# B&R Automation Studio project TD52 (part 100)

#### gwt.var - Local variables
```iecst
VAR
	xGR_MAXR_FA_AN_LAGA1 : GR_MAXR;
	xGR_MAXR_FA_GWW1 : GR_MAXR;
	xGR_MAXR_FA_AN_LAGW2 : GR_MAXR;
	xGR_MAXR_FA_AN_LAGW1 : GR_MAXR;
	xGR_MAXR_FA_AN_GW_TA : GR_MAXR := (0);
	xGR_MAXR_FA_AN_LAGA2 : GR_MAXR;
	xGR_MAXR_FA_GWW2 : GR_MAXR;
	xGR_MAXR_FA_GWA3 : GR_MAXR;
	xGR_MAXR_FA_GWA2 : GR_MAXR;
	xGR_MAXR_FA_GWW3 : GR_MAXR;
	xGR_MAXR_FA_GWA1 : GR_MAXR;
	xTON_FA_T_AN_LAGW1 : TON;
	xTON_FA_T_AN_LAGA1 : TON;
	xTON_FA_T_AN_GWA3 : TON;
	xTON_FA_T_AN_LAGA2 : TON;
	xTON_FA_T_AN_GWA2 : TON;
	xTON_FA_AN_GWTA : TON;
	xTON_FA_T_AN_GWA1 : TON;
	xTON_FA_AN_GWW2 : TON;
	xTON_FA_AN_GWW3 : TON;
	xTON_FA_AN_GWW1 : TON;
	xTON_FA_T_AN_LAGW2 : TON;
	xTON_FA_AN_GWTW : TON := (0);
	xGR_MAXR_FA_AN_GW_TW : GR_MAXR := (0);
END_VAR
```

### Program Logical/Generator/pf_ctr (IEC, version 4.14.0) - power factor control

#### pf_ctrCyclic.st
```iecst
(*******************************************************************************
pf_ctr - power factor control
		 power reduction due to voltage or frequency deviation

This code is confidential and proprietary to the INNIO Company.
It may not be used in any form, or reproduced in any manner, without the express
written permission of the INNIO Company.
Copyright, INNIO Company, 2019

Customized modifications: -
------------------------

History:
-------
0.10	30-05-2008	Gföller,	generated
		10-02-2009	Gföller,	calculation for Q- limit rQ_LIM added
		11-02-2009	Gföller,	calculation of limit added
		07-04-2009	Gföller,	correction of scale of external limit
2.50.1	23-06-2009  Wasserer+Le	redesign, var7 customized connection, correction of limitations
		01-07-2009	lettenb.	f_deltaU_PROM added (bewertung U-abweichung)
2.60.0 12.08.2009	lettenb.	pf_contr rename to pf_ctr, task QP_red included into pf_ctr
								PFSollext, ssPFext1-3fix, selPFext1-3fix added (from pf_cust)
					Tinello		delete Para.rPF_CosPCtr_Ext_Pnt1 and ssPf_P2 from Init / changed reg8 into reg13
					lettenb.	power reduction by winding temperature: calc.error corr.
		14.10.2009				OUT_GC.rPF_GenCtr_Act:=1000 if IN_GC.gcb=off for controller X display
3.20.0	30.09.2010	Maier(BuR)	GS_EIN replaced with IN_GC.bGCB_On
3.30.0  10.10.2011	lettenb.	ssPowRedGenTemp: not active in case of M_MSGWT(sensor failure)
		28.10.2011	Tinello		usFreqNenn[1] / 10 --> parameter "nominal frequency" was increased by factor 10
		04.11.2011	lettenb.	M_MS_PFset added (limit PFset in case of MS)
4.02.0	14.05.2014	lettenb.	xTON_ErregAusf: Para.tiPF_CosPCtr_del --> Para.rTi_Q_MinDel, visu new version!
4.02.1	19.05.2014	lettenb.	control mode 4: scaling changed, bugfix
		27.05.2014	lettenb.	2156, 2157: MM2VIS.bMsg215x -> bMsg215x, moved TO MsgGC
		12.06.2014				set PFSoll_lin TO cosphi 1.0 in CASE OF MS failure, bugfix
		26.09.2014				ramp FOR u/f/T-gen.Pred changed acc.xt3 behavior
4.02.2  28.10.2014	lettenb.	rT_Gen_Wind_Max: > --> >= reduction interrupts IF 2 gen.wind.temp.are equal
		03.11.2014				cap.PF reduction, limitation PF reduction, bugfix
4.04.0	01.08.2016				cosphi limits removed -> 0.0 underexcited - 1 - 0.0 overexcited, Q_Set_AVR -> UNITROL (//LE)
4.05.0  30.11.2017	lettenb.	GR redesign, PF control -> Q control, write parameter removed(code guide line)
4.07.0	17.12.2018	lettenb.	Qlimitation by under voltage added
		22.05.2019	lettenb.	Qlimitation by gen.wind.temp.high, enable manuell settings with active rQ_Lim_T_GenWind, bugfix
4.09.0	18.11.2019	lettenb.	rU_Gen_Nom_2 substituted by  rU_Gen_Nom[1], rU_Gen_Nom_2 removed, (gridcode/lukas)
4.14.0	29.11.2024	Farre,		calculation of power reduction due to CosPhi <1, from OP to GC (issue #1700)

Instructions for use:
--------------------

Description:
------------
Q-control:
pf_ctr:
power reduction by under- or over voltage enabled
power reduction by under- or over frequency
power reduction by winding temperature high
power factor limitation by winding temperature high
power factor limitation by polar wheel angel
calculation of reactive power limit for loss of excitation(A1109)
selection point of control
pf_set from timetable GC -> GR: OUT_GC.rPF_Set_TimeTable
limiter out: rQ_Set_Lim -> pf_cust

pf_cust:
summation Q_set + Ctr_Q_out.y
generation operation status depending setpoints (idle mode, synch-mode, island volt.control)
operation status depending selection of setpoint
scaling for V/mA AO for old AVR (PF_set signal)
scaling for V    AO for UNITROL (Q_set)

Outstandings:
------------
*********************************************************************************)
PROGRAM _CYCLIC

	(* begin program - QP reduction *)

	(* calculation of nominal power in parts per thousand *)
	rP_Gen_ppt	:= 1.000;

	(* power reduction by under- or over voltage enabled *)
	IF xOpMode.NetP AND Para.bPF_CosPCtr_U_Ena THEN

		(* calculation of voltage in parts per thousand HIGHER RESOLUTION FOR LOW VOLTAGE *)
		IF Para.rU_Gen_Nom[1] <> 0.0 AND Para.rU_Gen_Nom[1] <= 1000 THEN
			rU_AI_Gen_Avg_ppt	:= IN_GC.tU_Avg[1].Ai / Para.rU_Gen_Nom[1];

			(* scaling low voltage *)
			xSigScal_SpgRedLow(X:= rU_AI_Gen_Avg_ppt, X1:= Para.rPF_CosPCtr_U_Lo_End, Y1:= Para.rP_CosPCtr_U_Lo, X2:= Para.rPF_CosPCtr_U_Lo_Start, Y2:= 1.00);
			(* scaling high voltage *)
			xSigScal_SpgRedHigh(X:= rU_AI_Gen_Avg_ppt, X1:= Para.rPF_CosPCtr_U_Hi_Start, Y1:= 1.00,	X2:= Para.rPF_CosPCtr_U_Hi_End, Y2:= Para.rP_CosPCtr_U_Hi);

		END_IF;

		(* calculation of voltage in parts per thousand *)
		IF Para.rU_Gen_Nom[1] <> 0.0 AND Para.rU_Gen_Nom[1] > 1000 THEN
			rU_AI_Gen_Avg_ppt	:= IN_GC.tU_Avg[1].Ai / Para.rU_Gen_Nom[1];

			(* scaling low voltage *)
			xSigScal_SpgRedLow(X:= rU_AI_Gen_Avg_ppt, X1:= Para.rPF_CosPCtr_U_Lo_End, Y1:= Para.rP_CosPCtr_U_Lo, X2:= Para.rPF_CosPCtr_U_Lo_Start, Y2:= 1.00);
			(* scaling high voltage *)
			xSigScal_SpgRedHigh(X:= rU_AI_Gen_Avg_ppt, X1:= Para.rPF_CosPCtr_U_Hi_Start, Y1:= 1.00,	X2:= Para.rPF_CosPCtr_U_Hi_End,	Y2:= Para.rP_CosPCtr_U_Hi);

		END_IF;

		(* reduction active *)
		IF xSigScal_SpgRedLow.Y_SCAL < 1.00 THEN			(* power reduction by low voltage *)
			rP_CosPCtr_U_Red           := xSigScal_SpgRedLow.Y_SCAL;
			OUT_GC.bP_Red_CosPCtr_U_Lo := TRUE;
		ELSIF xSigScal_SpgRedHigh.Y_SCAL < 1.00 THEN		(* power reduction by high voltage *)
			rP_CosPCtr_U_Red           := xSigScal_SpgRedHigh.Y_SCAL;
			OUT_GC.bP_Red_CosPCtr_U_Hi := TRUE;
		ELSE
			rP_CosPCtr_U_Red	       := 1.00;
			OUT_GC.bP_Red_CosPCtr_U_Lo := FALSE;
			OUT_GC.bP_Red_CosPCtr_U_Hi := FALSE;
		END_IF;
	ELSE
		rP_CosPCtr_U_Red	       := 1.00;
		OUT_GC.bP_Red_CosPCtr_U_Lo := FALSE;
		OUT_GC.bP_Red_CosPCtr_U_Hi := FALSE;
 	END_IF;

	(* power reduction by under- or over frequency enabled *)
	IF (xOpMode.NetP) THEN	(* function for frequency too low always enabled *)

		(* calculation of frequency in parts per thousand *)
		IF Para.rF_Nom[1] > 0.0 THEN
			rF_Gen_ppt	:= IN_GC.tF_MMD[1].Ai / Para.rF_Nom[1];
		END_IF;

		(* frequency too low *)
		xSigScal_FrqRedLow(X:= rF_Gen_ppt, X1:= Para.rPF_CosPCtr_F_Lo_End, Y1:= Para.rP_CosPCtr_F_Lo, X2:= Para.rPF_CosPCtr_F_Lo_Start, Y2:= 1.00);
		(* frequency too high *)
		IF Para.bPF_CosPCtr_F_Ena THEN		(* function for frequency too high enabled by parameter *)
			xSigScal_FrqRedHigh(X:= rF_Gen_ppt, X1:= Para.rPF_CosPCtr_F_Hi_Start, Y1:= 1.00, X2:= Para.rPF_CosPCtr_F_Hi_End, Y2:= Para.rP_CosPCtr_F_Hi);
		END_IF;

		(* reduction active *)
		IF xSigScal_FrqRedLow.Y_SCAL < rP_Gen_ppt THEN								        (* power reduction by low frequency *)
			rP_CosPCtr_F_Red           := xSigScal_FrqRedLow.Y_SCAL;
			OUT_GC.bP_Red_CosPCtr_F_Lo := TRUE;
		ELSIF Para.bPF_CosPCtr_F_Ena AND xSigScal_FrqRedHigh.Y_SCAL < rP_Gen_ppt THEN		(* power reduction by high frequency *)
			rP_CosPCtr_F_Red           := xSigScal_FrqRedHigh.Y_SCAL;
			OUT_GC.bP_Red_CosPCtr_F_Hi := TRUE;
		ELSE
			rP_CosPCtr_F_Red    := 1.00;
			OUT_GC.bP_Red_CosPCtr_F_Lo := FALSE;
			OUT_GC.bP_Red_CosPCtr_F_Hi := FALSE;
		END_IF;

		(* hysteresis window for over frequency *)
		IF ((IN_GC.tF_MMD[1].Ai > Para.rF_Nom[1]) AND Para.bPF_CosPCtr_F_Ena) THEN	(* frequency higher than nominal frequency *)
  			IF rF_Gen_ppt > Para.rPF_CosPCtr_F_Hi_Start THEN		(* frequency higher than limit for over frequency *)
				IF rP_CosPCtr_F_Red < ssPowRedFrqMin THEN
					ssPowRedFrqMin := rP_CosPCtr_F_Red;		(* remember minimum power *)
				END_IF
			END_IF

			IF rF_Gen_ppt < Para.rPF_CosPCtr_F_ret THEN		(* frequency returns to normal frequency *)
	  			ssPowRedFrqMin := 1.00;
			END_IF

			rP_CosPCtr_F_Red := ssPowRedFrqMin;
		END_IF
	ELSE
		rP_CosPCtr_F_Red	       := 1.00;
		OUT_GC.bP_Red_CosPCtr_F_Lo := FALSE;
		OUT_GC.bP_Red_CosPCtr_F_Hi := FALSE;
 	END_IF;

	(* power factor limitation by winding temperature high *)
	IF Para.bT_Gen_Wind_Ena THEN		(* monitoring only when PT100 for winding temperature are used *)
		(* determination of maximum winding temperature *)
		IF 		((IN_GC.tT_Gen_Wind_Act_L1.Ai >= IN_GC.tT_Gen_Wind_Act_L2.Ai)
			AND  (IN_GC.tT_Gen_Wind_Act_L1.Ai >= IN_GC.tT_Gen_Wind_Act_L3.Ai)
			AND   IN_GC.tT_Gen_Wind_Act_L1.GoodQual) THEN
  			rT_Gen_Wind_Max := IN_GC.tT_Gen_Wind_Act_L1.Ai;
		ELSIF  ((IN_GC.tT_Gen_Wind_Act_L2.Ai >= IN_GC.tT_Gen_Wind_Act_L1.Ai)
			AND (IN_GC.tT_Gen_Wind_Act_L2.Ai >= IN_GC.tT_Gen_Wind_Act_L3.Ai)
			AND  IN_GC.tT_Gen_Wind_Act_L2.GoodQual) THEN
  			rT_Gen_Wind_Max := IN_GC.tT_Gen_Wind_Act_L2.Ai;
		ELSIF  ((IN_GC.tT_Gen_Wind_Act_L3.Ai >= IN_GC.tT_Gen_Wind_Act_L1.Ai)
			AND (IN_GC.tT_Gen_Wind_Act_L3.Ai >= IN_GC.tT_Gen_Wind_Act_L2.Ai)
			AND IN_GC.tT_Gen_Wind_Act_L3.GoodQual) THEN
			rT_Gen_Wind_Max := IN_GC.tT_Gen_Wind_Act_L3.Ai;
		ELSE
			rT_Gen_Wind_Max := 0.0;
		END_IF

		IF Para.bPF_CosPCtr_Ena THEN		(* if power factor controller is enabled *)
			(* reduction of power factor by winding temperature *)
			IF rT_Gen_Wind_Max  >= Para.rPF_CosPCtr_T_max AND Para.rPF_CosPCtr_T_red > 0.0 THEN
				IF NOT bPF_Once THEN
					ssPF_Begin	:= IN_GC.tPF_Act[1].Ai; (* value: -0.7 bis -1.0 = cap., 0.7 bis 1.0 = ind *)
	   				bPF_Once := TRUE;
				END_IF;

				IF ssPF_Begin >= 0 THEN	(* ind *)
					rPF_CosPCtr_T_Lim := ssPF_Begin + ((rT_Gen_Wind_Max - Para.rPF_CosPCtr_T_max) * Para.rPF_CosPCtr_T_red);
					IF rPF_CosPCtr_T_Lim > 1.0 THEN	rPF_CosPCtr_T_Lim := 1.0;(* limit calculation to PF = 1 *)
					END_IF;
				ELSE	                (* cap *)
					rPF_CosPCtr_T_Lim := ssPF_Begin - ((rT_Gen_Wind_Max - Para.rPF_CosPCtr_T_max) * Para.rPF_CosPCtr_T_red);
					IF rPF_CosPCtr_T_Lim < -1.0 THEN rPF_CosPCtr_T_Lim := 1.0;(* limit calculation to PF = 1 *)
					END_IF;
				END_IF;

			ELSE
				bPF_Once := FALSE;
				IF IN_GC.tPF_Act[1].Ai > 0.0 THEN rPF_CosPCtr_T_Lim :=  0.001; (* no limit for PF *)//LE
				ELSE                              rPF_CosPCtr_T_Lim := -0.001;
				END_IF;
			END_IF;
		ELSE
			IF IN_GC.tPF_Act[1].Ai > 0.0 THEN rPF_CosPCtr_T_Lim :=  0.001; (* no limit for PF *)//LE
			ELSE                              rPF_CosPCtr_T_Lim := -0.001;
			END_IF;
		END_IF;

		(* power reduction by winding temperature *)
		IF rT_Gen_Wind_Max >= Para.rP_CosPCtr_T_Hi AND rT_Gen_Wind_Max  <> 0 THEN
			rP_CosPCtr_T_Red := 1.00 - ((rT_Gen_Wind_Max - Para.rP_CosPCtr_T_Hi) * Para.rPF_CosPCtr_T_wind);
		ELSE
			rP_CosPCtr_T_Red := 1.00;
		END_IF
	ELSE
		rP_CosPCtr_T_Red := 1.00;
	END_IF

	rP_CosPCtr_U_Red := LIMIT(0.50, rP_CosPCtr_U_Red, 1.00);
	rP_CosPCtr_F_Red := LIMIT(0.50, rP_CosPCtr_F_Red, 1.00);
	rP_CosPCtr_T_Red := LIMIT(0.50, rP_CosPCtr_T_Red, 1.00);

	(* calculation of power reduction *)
	IF IN_GC.rP_Nom <> 0.0 THEN

		(* generator voltage *)
		IF rP_CosPCtr_U_Red < 1.00 THEN
	 		rP_CosPCtr_U_Red := (IN_GC.rP_Nom - ((1.00-rP_CosPCtr_U_Red) * IN_GC.rP_Nom / 1.00)) / IN_GC.rP_Nom;
		ELSE
			rP_CosPCtr_U_Red := IN_GC.rP_Nom / IN_GC.rP_Nom;
		END_IF;

		(* generator frequency *)
		IF rP_CosPCtr_F_Red < 1.00 THEN
	 		rP_CosPCtr_F_Red := (IN_GC.rP_Nom - ((1.00-rP_CosPCtr_F_Red) * IN_GC.rP_Nom / 1.00)) / IN_GC.rP_Nom;
		ELSE
			rP_CosPCtr_F_Red := IN_GC.rP_Nom / IN_GC.rP_Nom;
		END_IF;

		(* generator winding temperature *)
		IF rP_CosPCtr_T_Red < 1.00 THEN
	 		rP_CosPCtr_T_Red := (IN_GC.rP_Nom - ((1.00-rP_CosPCtr_T_Red) * IN_GC.rP_Nom / 1.00))/ IN_GC.rP_Nom;
		ELSE
			rP_CosPCtr_T_Red := IN_GC.rP_Nom / IN_GC.rP_Nom;
		END_IF;

	ELSE
		(* Set lowest value in case of a rP_Nom value is zero *)
		rP_CosPCtr_T_Red := 0.5;
		rP_CosPCtr_F_Red := 0.5;
		rP_CosPCtr_U_Red := 0.5;
	END_IF;

	(* smoother transition *)
	xRAMPE_RedGenSpg(enable:= IN_GC.tGCB_On.Di, In:= rP_CosPCtr_U_Red, Rise:= 0.007, Sink:= 0.007, TC_Time:= 100);(* 0.007: 100->50% ca.35" *)
	xRAMPE_RedGenSpg();
	rP_CosPCtr_U_Red	:= xRAMPE_RedGenSpg.Out;

	xRAMPE_RedGenFrq(enable:= IN_GC.tGCB_On.Di, In:= rP_CosPCtr_F_Red, Rise:= 0.007, Sink:= 0.007, TC_Time:= 100);
	xRAMPE_RedGenFrq();
	rP_CosPCtr_F_Red  := xRAMPE_RedGenFrq.Out;

	xRAMPE_RedGenTemp(enable:= IN_GC.tGCB_On.Di, In:= rP_CosPCtr_T_Red, Rise:= 0.007, Sink:= 0.007, TC_Time:= 100);
	xRAMPE_RedGenTemp();
	rP_CosPCtr_T_Red	:= xRAMPE_RedGenTemp.Out;

(*-----------------------------------------------------------------------------------*)
	(* CALCULATION OF REACTIVE POWER LIMIT - polar wheel angle                       *)
	(* calculation of auxiliary variables for reactive power *)
	bU_Gen_Norm := IN_GC.tEng_Run.Do AND IN_GC.tGCB_On.Di AND NOT IN_GC.tGen_Exc_Off.Di;
	IF bU_Gen_Norm AND NOT (IN_GC.bTP_GrC_Event AND (IN_GC.tU_Avg[1].Ai < (Para.rU_Gen_Nom[1] * 0.5))) THEN
		rFact1	:= IN_GC.tU_Avg[1].Ai * IN_GC.tU_Avg[1].Ai * Para.rS_Nom;
	ELSE
		rFact1	:= Para.rU_Gen_Nom[1] * Para.rU_Gen_Nom[1] * Para.rS_Nom;
 	END_IF;
	rFact2	:= Para.rU_Gen_Nom[1] * Para.rU_Gen_Nom[1];

	(* calculation of reactive power limitation of polar wheel angle (Polradwinkel)  *)
	rDeltaRAD	:= Para.rAng_CosPCtr_Lim / (180.0 / rCnst_PI);	(* conversion in radian measure (Bogenmaß) *)
	IF 	TAN(rDeltaRAD) <> 0 AND (Para.rxd_CosPCtr * rFact2) <> 0 THEN	(* avoid zero division *)
		rAng_CosPCtr_LimCalc := IN_GC.tP_Act[1].Ai / TAN(rDeltaRAD) - rFact1 / (Para.rxd_CosPCtr * rFact2);

		rPF_CosPCtr_MinCalc1 := 0.0 / TAN(rDeltaRAD) - rFact1 / (Para.rxd_CosPCtr * rFact2);
		rPF_CosPCtr_MinCalc2 := IN_GC.rP_Nom / TAN(rDeltaRAD) - rFact1 / (Para.rxd_CosPCtr * rFact2);
	END_IF;

	(* calculation of reactive power limitation for LOSS OF EXCITATION  *)
	rDelta_TripRAD	:= Para.rAng_CosPCtr_Min / (180.0 / rCnst_PI);	(* conversion in radian measure (Bogenmaß) *)
	IF 	TAN(rDelta_TripRAD) <> 0 AND (Para.rxd_CosPCtr * rFact2) <> 0 THEN	(* avoid zero division *)
		rAng_CosPCtr_MinCalc := IN_GC.tP_Act[1].Ai  / TAN(rDelta_TripRAD) - rFact1 / (Para.rxd_CosPCtr * rFact2);

		rPF_CosPCtr_LimCalc1 := 0.0 / TAN(rDelta_TripRAD) - rFact1 / (Para.rxd_CosPCtr * rFact2);
		rPF_CosPCtr_LimCalc2 := IN_GC.rP_Nom / TAN(rDelta_TripRAD) - rFact1 / (Para.rxd_CosPCtr * rFact2);
	END_IF;

	IF rAng_CosPCtr_LimCalc <= rAng_CosPCtr_MinCalc THEN
 		rAng_CosPCtr_LimCalc :=	rAng_CosPCtr_MinCalc;
	END_IF;

	(* LOSS OF EXCITATION AMM 1109 *)
	xTON_ErregAusf.IN := (IN_GC.tQ_Act[1].Ai  < rAng_CosPCtr_MinCalc) AND IN_GC.tPB2MM.bParaSetupOk; (* generator reactive power > limit value *)
	xTON_ErregAusf.PT := REAL_TO_TIME(Para.rTi_Q_MinDel[1] *1000); (* 0.1sec * 1000 = ms *)
	xTON_ErregAusf();

	bPF_CosPCtr_Trip	:= xTON_ErregAusf.Q; (* delay loss of excitation *)

	(* END CALCULATION OF REACTIVE POWER LIMIT 			END CALCULATION OF REACTIVE POWER LIMIT  *)
	(* ==================================================================================================== *)

	(*-----------------------------------------------------------------------------------*)
	(* CALCULATION OF REACTIVE POWER LIMIT by under voltage *)
	(* calculation of auxiliary variables for reactive power *)
//			Para.bQ_UnderExc_Ena
//	Uact	IN_GC.tU_Avg[1].Ai			[V]
//	Qmin1	Para.rQ_UnderExc_Lim 	-27	[%]
//	Umin1	Para.rQ_UnderExc_Start	95	[%]
//	Umin2	Para.rQ_UnderExc_Stop	90	[%]
//	Qmin2	Para.rQ_UnderExc_Lim2	0	[%]  Qmin2 have to be higher then Qmin
	IF Para.rU_Gen_Nom[1] > 0.0 THEN rUact := IN_GC.tU_Avg[1].Ai / Para.rU_Gen_Nom[1];
	END_IF;

	IF    rUact > Para.rQ_UnderExc_Start THEN rQmin_U := Para.rQ_UnderExc_Lim;
	ELSIF rUact < Para.rQ_UnderExc_Stop  THEN rQmin_U := MAX(Para.rQ_UnderExc_Lim2, Para.rQ_UnderExc_Lim);(* Qmin2 have to be higher then Qmin *)
	ELSE  xSigScal_Qlim_Ulow(X:= rUact, X1:= Para.rQ_UnderExc_Start, Y1:= Para.rQ_UnderExc_Lim, X2:= Para.rQ_UnderExc_Stop, Y2:= MAX(Para.rQ_UnderExc_Lim2, Para.rQ_UnderExc_Lim));
		  rQmin_U := xSigScal_Qlim_Ulow.Y_SCAL;(* U too low *)
//		  rUact_Umin2 := rUact - Para.rQ_UnderExc_Stop;(* for testing *)
//		  rUmin1_Umin2 := ABS(Para.rQ_UnderExc_Start) - ABS(Para.rQ_UnderExc_Stop);
//		  rQmin2_Qmin1 := ABS(Para.rQ_UnderExc_Lim2) - ABS(Para.rQ_UnderExc_Lim);
//		  rQmin_U := (rUact_Umin2 * (rQmin2_Qmin1 / rUmin1_Umin2)) + Para.rQ_UnderExc_Lim2; (*[%]*)
	END_IF;

//	(* END CALCULATION OF REACTIVE POWER LIMIT 			END CALCULATION OF REACTIVE POWER LIMIT  *)
//	(* ==================================================================================================== *)

	(* ==================================================================================================== *)
	(* SELECTION POINT OF CONTROL                                                                           *)
       (* defines the point of control for Q, PF or U *)
	(*  0:	customized AI *)
	(*  1:	MMU1 generator *)
	(*	2:	MMU2 point of connection *)
	(*  3:  direct control *)

		CASE Para.iQ_GrC_PointCtrl OF
			0:	rS_POC_Act  := IN_GC.rS_POC_Act_Cust;	(* customized/c_statGR *)
				rP_POC_Act  := IN_GC.rP_POC_Act_Cust;
				rQ_POC_Act  := IN_GC.rQ_POC_Act_Cust;
				rPF_POC_Act	:= IN_GC.rPF_POC_Act_Cust;
				rU_POC_Act  := 0;						(* not used *)

			1:	rS_POC_Act  := IN_GC.tS_Act[1].Ai;		(* MMU1/generator *)
				rP_POC_Act  := IN_GC.tP_Act[1].Ai;
				rQ_POC_Act  := IN_GC.tQ_Act[1].Ai;
				rPF_POC_Act	:= IN_GC.tPF_Act[1].Ai;
				rU_POC_Act  := IN_GC.tU_Avg[1].Ai;

			2:	rS_POC_Act  := IN_GC.tS_Act[2].Ai;		(* MMU2/point of connection *)
				rP_POC_Act  := IN_GC.tP_Act[2].Ai;
				rQ_POC_Act  := IN_GC.tQ_Act[2].Ai;
				rPF_POC_Act	:= IN_GC.tPF_Act[1].Ai;
				rU_POC_Act  := IN_GC.tU_Avg[2].Ai;

		    3:	rS_POC_Act  := IN_GC.tS_Act[1].Ai;		(* MMU1/generator *)
				rP_POC_Act  := IN_GC.tP_Act[1].Ai;
				rQ_POC_Act  := IN_GC.tQ_Act[1].Ai;
				rPF_POC_Act	:= IN_GC.tPF_Act[1].Ai;
				rU_POC_Act  := IN_GC.tU_Avg[1].Ai;

				ELSE
				rS_POC_Act  := 0;
				rP_POC_Act  := 0;
				rQ_POC_Act  := 0;
				rPF_POC_Act	:= 1;
				rU_POC_Act  := 0;
		END_CASE;

		IF xOpMode.NetP AND Para.rS_Nom > 0 AND IN_GC.rP_Nom > 0 AND Para.rS_Nom > IN_GC.rP_Nom THEN
			rS_POC_Act_Norm := rS_POC_Act / Para.rS_Nom;
			rP_POC_Act_Norm := rP_POC_Act / IN_GC.rP_Nom;
			rQ_POC_Act_Norm := rQ_POC_Act / Para.rS_Nom;
		END_IF;

		(* linearization rPF_POC_Act *)
		(* +0,7(ind/overexc.)..1,0..-0,7(cap/underexc.) ==> 0,70 .. 1,00 .. 1,30 *)
		//Filterung des Cos(PHI) Signals
		IF rPF_POC_Act >= 0 THEN rPF_Act_lin := rPF_POC_Act;
		ELSE					 rPF_Act_lin := rPF_POC_Act + 2.000;
		END_IF;
		xFILTER_PF(In := rPF_Act_lin, Filter := 10);

		MM2VIS.rPF_POC_Act_lin	:= xFILTER_PF.Out;

		(* diagram Y(graph)-value point of control (POC)*)
		IF Para.rS_Nom > 0 THEN
			MM2VIS.rQS_POC := rQ_POC_Act / Para.rS_Nom;
		END_IF;

		(* ==================================================================================================== *)
		(* selection of set point by time table from parameters -> GR *)
		(*
		time frame 1		begin- hour 1/ begin- minute 1	till	stop- hour 1/ stop- minute 1
							stop- hour 2/ stop- minute 2 := begin- hour 1/ begin- minute 1
		time frame 2		begin- hour 2/ begin- minute 2	till	stop- hour 2/ stop- minute 2
							stop- hour 3/ stop- minute 3 := begin- hour 2/ begin- minute 2
	.
		. *)
		(* getting time of the controller *)
		DTGetTime_RPS.enable := TRUE;							(* getting *)
		DTGetTime_RPS();
		DT_TO_DTStructure(DTGetTime_RPS.DT1, ADR(tRealTime));	(* change format *)
		DTGetTime_RPS.status;

		IF  tRealTime.hour >= REAL_TO_USINT(Para.rPF_CosPCtr_h[0]) AND tRealTime.minute >= REAL_TO_USINT(Para.rPF_CosPCtr_m[0]) THEN
			rPF_TimeAct := Para.rPF_CosPCtr_Tme_Set[0];
		END_IF
		IF  tRealTime.hour >= REAL_TO_USINT(Para.rPF_CosPCtr_h[1]) AND tRealTime.minute >= REAL_TO_USINT(Para.rPF_CosPCtr_m[1]) THEN
			rPF_TimeAct := Para.rPF_CosPCtr_Tme_Set[1];
		END_IF
		IF  tRealTime.hour >= REAL_TO_USINT(Para.rPF_CosPCtr_h[2]) AND tRealTime.minute >= REAL_TO_USINT(Para.rPF_CosPCtr_m[2]) THEN
			rPF_TimeAct := Para.rPF_CosPCtr_Tme_Set[2];
		END_IF
		IF  tRealTime.hour >= REAL_TO_USINT(Para.rPF_CosPCtr_h[3]) AND tRealTime.minute >= REAL_TO_USINT(Para.rPF_CosPCtr_m[3]) THEN
			rPF_TimeAct := Para.rPF_CosPCtr_Tme_Set[3];
		END_IF
		IF  tRealTime.hour >= REAL_TO_USINT(Para.rPF_CosPCtr_h[4]) AND tRealTime.minute >= REAL_TO_USINT(Para.rPF_CosPCtr_m[4]) THEN
			rPF_TimeAct := Para.rPF_CosPCtr_Tme_Set[4];
		END_IF
		IF  tRealTime.hour >= REAL_TO_USINT(Para.rPF_CosPCtr_h[5]) AND tRealTime.minute >= REAL_TO_USINT(Para.rPF_CosPCtr_m[5]) THEN
			rPF_TimeAct := Para.rPF_CosPCtr_Tme_Set[5];
		END_IF

		OUT_GC.rPF_Set_TimeTable := rPF_TimeAct;	(* GC -> GR *)(* + = overexited/ind., - = underexited/cap. *)

		(* Limited rQSoll_Lim_GR2GC from GR -> GC *)
		IN_GC.rQSoll_Lim_GR2GC;		(* including limitation from Q(U) and QLim_Ext *)

	(* ==================================================================================================== *)
	(* Q limit by winding temperature *)
		(* umrechnung rPF_CosPCtr_T_Lim -> rQ_Lim_T_GenWind[%] *)
		IF Para.bT_Gen_Wind_Ena AND Para.bPF_CosPCtr_Ena AND xOpMode.NetP AND IN_GC.rP_Act_Norm_Filt > 0.10 AND rPF_CosPCtr_T_Lim <> 0.000 THEN
			IF    rPF_CosPCtr_T_Lim > 0.000 THEN rQ_Lim_T_GenWind :=        IN_GC.rP_Act_Norm_Filt * 0.8 * (SQRT(1 / (rPF_CosPCtr_T_Lim * rPF_CosPCtr_T_Lim) -1));
			ELSIF rPF_CosPCtr_T_Lim < 0.000 THEN rQ_Lim_T_GenWind := (-1) * IN_GC.rP_Act_Norm_Filt * 0.8 * (SQRT(1 / (rPF_CosPCtr_T_Lim * rPF_CosPCtr_T_Lim) -1));
			END_IF;
		ELSE
			IF IN_GC.rQSoll_Lim_GR2GC >= 0.0 THEN rQ_Lim_T_GenWind :=  1.0;
			ELSE                                  rQ_Lim_T_GenWind := -1.0;
			END_IF;
		END_IF;

		(*------------------------------------------------------------------------------------------------------*)
		(* Q-limit by polar wheel angle *)
		(* umrechnung Q_Lim_PWA[kVAr] -> rQ_Lim_PWA[%] *)
		IF Para.rS_Nom > 0 AND xOpMode.NetP AND IN_GC.rP_Act_Norm_Filt > 0.10 THEN
			rQ_Lim_PWA := rAng_CosPCtr_LimCalc / Para.rS_Nom;                      (* pos. = uebererregt = ind.Q-abgabe/plant *)
 		ELSE																	   (* neg. = untererregt = kap.Q-abgabe/plant *)
			rQ_Lim_PWA := -1.0;
		END_IF;

		(*------------------------------------------------------------------------------------------------------*)
		(* Q-limit by under voltage (under excitation) *)
		IF Para.bQ_UnderExc_Ena AND xOpMode.NetP AND IN_GC.rP_Act_Norm_Filt > 0.10 THEN
			rQ_Lim_U := rQmin_U;(* [%] *)
 		ELSE																	   (* neg. = untererregt = kap.Q-abgabe/plant *)
			rQ_Lim_U := -1.0;
		END_IF;
		(*------------------------------------------------------------------------------------------------------*)
		(* LIMITER *)
		rQ_Set_Lim        := IN_GC.rQSoll_Lim_GR2GC; (* limiter in *)

		IF    bPF_Once AND ABS(IN_GC.rQSoll_Lim_GR2GC) > ABS(rQ_Lim_T_GenWind) THEN rQ_Set_Lim := rQ_Lim_T_GenWind;(* ind./overexcited/+kVAr *)
			bMsg2156   := TRUE; 		   (* B2156 Q-limit by gen.wind.temp.*)
		ELSIF bPF_Once AND ABS(IN_GC.rQSoll_Lim_GR2GC) < ABS(rQ_Lim_T_GenWind) THEN rQ_Set_Lim := IN_GC.rQSoll_Lim_GR2GC;
			bMsg2156   := TRUE; 		   (* B2156 Q-limit by gen.wind.temp.*)
		ELSE  					                                          bMsg2156   := FALSE;
		END_IF;

		IF IN_GC.tPF_Act[1].Ai < 0.0 AND IN_GC.rQSoll_Lim_GR2GC < rQ_Lim_PWA AND rQ_Set_Lim < rQ_Lim_PWA
																	 THEN rQ_Set_Lim := rQ_Lim_PWA;      (* cap./underexcited/-kVAr *)
																		  bMsg2157   := TRUE;            (* B2157 Q-limit by polar wheel angel *)
		ELSE		                                                      bMsg2157   := FALSE;
		END_IF;

		IF IN_GC.tPF_Act[1].Ai < 0.0 AND IN_GC.rQSoll_Lim_GR2GC < rQ_Lim_U AND rQ_Set_Lim < rQ_Lim_U
																	 THEN rQ_Set_Lim := rQ_Lim_U;        (* cap./underexcited/-kVAr *)
																		  bMsg2998   := TRUE;            (* B2998 Q-limit by under voltage *)
		ELSE		                                                      bMsg2998   := FALSE;
		END_IF;

		rQ_Set_Lim;	(* limiter out -> pf_Cust *)

		MM2VIS.bQ_Lim_On := MM2VIS.bSel_AVR_Set AND    (IN_GC.bQSetLim	(*GR*)
		                							OR  bMsg2156	    (*GC*)
		                							OR  bMsg2157	    (*GC*)
		                							OR  bMsg2998);	    (*GC*)

		(*------------------------------------------------------------------------------------------------------*)
		(*** GC-> OP: Power Reduction CosPhi < 1 ***)
			IF IN_GC.tPF_Act[1].Ai < 0.98 AND IN_GC.tPF_Act[1].Ai > 0 AND IN_GC.rP_Act_Norm_Filt > 0.25 AND IN_GC.tPB2MM.bParaSetupOk AND Para.rEta_Gen_PF08 < Para.rEta_Gen_PF1 AND IN_GC.tGCB_On.Di THEN
				IF Para.rEta_Gen_PF1 <> 0 THEN
					rP_Red_Eta_Gen_Norm_int :=	(IN_GC.tPF_Act[1].Ai - 0.8) / (0.98 - 0.8)
										*	(1.0 - Para.rEta_Gen_PF08 / Para.rEta_Gen_PF1)
										+	Para.rEta_Gen_PF08 / Para.rEta_Gen_PF1;

				ELSE
					rP_Red_Eta_Gen_Norm_int := 1.0;
				END_IF
			ELSE
				rP_Red_Eta_Gen_Norm_int 	:= 1.0;
			END_IF

			xTON_rPRed(IN := (rP_Red_Eta_Gen_Norm_int < 1.0), PT := tDelayPRed);
			IF xTON_rPRed.Q THEN
				OUT_GC.rP_Red_Eta_Gen_Norm 	:= rP_Red_Eta_Gen_Norm_int;
			ELSE
				OUT_GC.rP_Red_Eta_Gen_Norm 	:= 1.0;
			END_IF;
		(*------------------------------------------------------------------------------------------------------*)

	(* ==================================================================================================== *)
	(* Werte für Regler und Anzeigen *)
	(* ==================================================================================================== *)

	RPS_s_oldQPF_XT := USINT_TO_UINT(tRealTime.second);

	OUT_GC.rP_Red_CosPCtr_F_Norm := rP_CosPCtr_F_Red;
	OUT_GC.rP_Red_CosPCtr_T_Norm := rP_CosPCtr_T_Red;
	OUT_GC.rP_Red_CosPCtr_U_Norm := rP_CosPCtr_U_Red;

END_PROGRAM
```

#### pf_ctrInit.st
```iecst
(*******************************************************************************
pf_ctr  Initialization

This code is confidential and proprietary to the INNIO Company.
It may not be used in any form, or reproduced in any manner,
without the express written permission of the INNIO Company.
Copyright, INNIO Company, 2019

Customized modifications: -
------------------------

History:
-------

********************************************************************)
PROGRAM _INIT

	ssPowRedFrqMin := 1.000;

	(* PVs not yet used *)
	PF_Out1;
	ssP_mains_scale1;
	PF_Out2;
	ssQ_mains_scale1;
	ssP_mains_scale2;
	bMI_MMU;
	ssQ_mains_scale2;
	bMIPCont_SPext;
	bPF_LIM_Temp;
	ssQ_mainsOffset;
	bMIPCont;
	ssMIRPCont_SP;
	ssMIPCont_SP;
	bMIRPCont_SPext;

END_PROGRAM
```

#### pf_ctr.var
```iecst
VAR
	rPF_CosPCtr_T_Lim : REAL := 0.0; (*Power factor limit by winding temperature limit*)
	rT_Gen_Wind_Max : REAL; (*Stores the maximum temperature of the 3 windings*)
	bPF_Once : BOOL;
	bU_Gen_Norm : BOOL;
	xRAMPE_RedGenTemp : RAMPE_R;
	xRAMPE_RedGenSpg : RAMPE_R;
	xRAMPE_RedGenFrq : RAMPE_R;
	ssPowRedFrqMin : REAL;
	rF_Gen_ppt : REAL;
	ssPF_Begin : REAL;
	rDelta_TripRAD : REAL;
	rFact1 : REAL;
	rFact2 : REAL;
	rPF_TimeAct : REAL;
	rDeltaRAD : REAL;
	xTON_ErregAusf : TON;
	RPS_s_oldQPF_XT : UINT;
	xSigScal_SpgRedHigh : xSigScal_R;
	xSigScal_FrqRedHigh : xSigScal_R;
	xSigScal_FrqRedLow : xSigScal_R;
	xSigScal_SpgRedLow : xSigScal_R;
	rQ_Lim_T_GenWind : REAL;
	rQ_Lim_PWA : REAL;
	xFILTER_PF : FILTER_R;
	rPF_Act_lin : REAL;
	rUact : REAL;
	xSigScal_Qlim_Ulow : xSigScal_R;
	rQmin_U : REAL;
	rQ_Lim_U : REAL;
	rP_Red_Eta_Gen_Norm_int : REAL := 1.0;	(*Power reduction due to Cosphi<1 calculated [p.u.]*)
	xTON_rPRed : TON; (*delay power reduction due to Cosphi<1 to OP*)
	tDelayPRed : TIME := T#200ms; (*delay power reduction due to Cosphi<1 [ms]*)
END_VAR
VAR CONSTANT
	rCnst_PI : REAL := 3.141593;
END_VAR
VAR
	DTGetTime_RPS : DTGetTime;
	tRealTime : DTStructure;
END_VAR
```

### Program Logical/Generator/pf_cust (IEC, version 4.12.0) - power factor custom

#### pf_custCyclic.st
```iecst
(*******************************************************************************
pf_cust 		Q-setpoint scaling for AVR

This code is confidential and proprietary to the INNIO Company.
It may not be used in any form, or reproduced in any manner,
without the express written permission of the INNIO Company.
Copyright, INNIO Company, 2022

Customized modifications: -
------------------------

History:
-------
V2.50.1	12.06.2009	Wasserer.	new
V2.60.0	12.08.2009	lettenb.	setpoint Umschaltung über kontakte transfered to pf_ctr
								(new parameter structure)
								task: reg_8gen(V2.50.2) included
					Tinello.	Changed reg8 into reg13
		27.10.2009	lettenb		bPF_AO_mA, AO_PF_gen removed
								separated outputs: OUT_GC.tPF_AO_PF_I, OUT_GC.rPF_AO_PF_U new
		30.11.2009	lettenb.	REG13.y := yBlock; ( ohne Rampe bei Block2 ) added
								(vermeidung von spannungsüberhöhungen bei umschaltung auf spgs.regler)
V3.20.0	24.03.2010	lettenb.	OUT_GC.rT_AO_Gen_T_In	added (UNITROL internal gen.power limitation)
		07.12.2010				u_offset_mA,u_offset_V added for v_matching
V3.99.9 13.02.2014  ganguly	    changed:
									 1. tPF_AO_PF_U to rPF_AO_PF_U
 									 2. tPF_AO_PF_I to rPF_AO_PF_I
									 3.	tCtrGenPF_Set to rCtrGenPF_Set
								These signals will be used as input to grid module and set from there
								because Grid module has priority over the AVR setpoint.
V4.01.0	14.05.2014	Denk		Bugfix, Intake air temp. for generator controller
					lettenb.	missing scaling added(acc.a_v3500) for user spec.signal correction
								missing rU_Gen_Diff_Match_U added(acc.a_v3500)
V4.01.1 06.03.2015	lettenb.	920, Para.bT_GenAirIn_Active added
V4.03.0	02.05.2016				xSigScal_PF.Y1: -0.700 -> +0.700, bugfix
V4.04.0	29.06.2016				tGen_T_In2.Ai, rP_Red_T_GenAirIn_Norm added, Dig142
        25.07.2016				tQ_AVR_Set_U.Ao: Q-vorgabe -> UNITROL,
								CtrGenPF: y-range 0-100% = 0,9kap. - 1 - 0,7ind. => 0,0kap. - 1 - 0,0ind.
		27.10.2016				rFactorU_Match removed, bugfix
		07.04.2017				rQ_AVR_Set: limitation FOR rPFSoll_lin_AVR added, TAN(ACOS(2-2) darf nicht 0 werden -> + unendlich, bugfix
V4.05.0 30.11.2017	lettenb.	GR redesign, PF control -> Q control
V4.05.1	15.03.2018				yBlock: fix 10 -> 2% Q, lastrampe bis aktivierung Q-controller, request vogl lukas
V4.07.0	03.06.2019	lettenb.	calc.rPF_POC_Set related to S_Nom(Lukas), set rPF_POC_Set := 1.0 in case of yBlock for PF control(DM110), bugfix
V4.12.0	05.12.2022	lettenb.	DIG142 Generator Air Inlet Temperature Power Reduction from: Tmax -> Tavg value of 2 sensors(QC1807)

Instructions for use:
--------------------

FUNCTION DIAGRAM:

+------------------------------------------------------------+
| Pred(U<>), Pred(f<>), Pred(Twind) ----------------------------------------> opstate
| PF_lim(Twind)                                              |
| Q_lim(PWA) polar wheel angel                               |
| PF_Timetable -------------------------------------------------------------> GR
+------------------------------------------------------------+
                              |
                              V
+------------------------------------------------------------+
| calculation PF_lim(Twind) -> QLim_Twind                    |
|                                                            |                GR
| depending on P_Act                                         |              +--------------------------------------------------+
|                                  IN_GC.rQSoll_filt_GR2GC[%] <---------------- OUT_GR.rQSoll_filt_GR2GC[%]                    |
|                                  IN_GC.rQSoll_lim_GR2GC [%] <---------------- OUT_GR.rQSoll_lim_GR2GC [%]                    |
|                                                            |              |   including limitation of Q(U) and QLim_External |
+------------------------------------------------------------+              +--------------------------------------------------+
                              | rQSoll_filt_GR2GC
                              V
                    +-------------------+
rQ_Lim_T_GenWind -->|      LIMITER      |
rQ_Lim_PWA       -->|                   |
rQ_Lim_PF        -->+-------------------+
                              |
                              V
                              |                                             +------------------------------------------------------+
                              |                                             | Block_CtrGenPF:                      (task: pf_cust) |
                              |                                             | - engine operation state(bPF_CosPCtr_block)          |
   +--------------------------+                                             |   rPF_CosPCtr_block                                  |
   |                                                                        +------------------------------------------------------+
   |                                                                        | U control(idle mode/synchroniz., rU_Gen_Diff_Match_U |
   |                                                                        +------------------------------------------------------+
   |          +-------------------------------------------------------+          |
   |          |   Ctr_Q(Reg33)                              direct    |          |
   v          |  +-----------+                              control   |          +
   rQ_Set_Lim-+--|\ W        |                                 \      v +         \
                 | )        Y|-------------------------------+  o---->0---------+  o--------------------- Q_AVR_Set_U.Ao
rQ_POC_Act_Norm -|/ X        | tCtr_Q_Out.Y                         +   rQ_Set_sum        rQ_AVR_Set
                 +-----------+

   Q_Set                      y       Q
    -1.0%(=-100%)          -1.0% = -100%                                             81.0 % Qnom = +8.16 V = cosphi 0.7  ind.
     0.0%(=   0%)           0.0% =    0%                                             60.0 % Qnom = +6.00 V = cosphi 0.8  ind.
    +1.0%(=+100%)          +1.0% = +100%                        overexcited          38.7 % Qnom = +3.87 V = cosphi 0.9  ind.
                                                               -------------------    0.0 % Qnom =  0.00 V = cosphi 1.0
                                                                underexcited        -26.3 % Qnom = -2.63 V = cosphi 0.95 cap.

												 +---------------------------------------+
												 | calculation rQ_AVR_Set -> rPF_POC_Set |
												 +---------------------------------------+
                                                                     |
                                                                     |  +------------+
                                                                     +--| scal. AO_V |-------PF_AO_PF_U  => AVR cosphi_setpoint +/-10V
                                                                     |  +------------+
                                                                     |                                 cosphi 0.0 ind. = +10.0 V
                                                                     |                                 cosphi 0.7 ind. =  +3.0 V = 20.0 mA
                                                                     |             overexcited         cosphi 0.8 ind. =  +2.0 V = 17.3 mA
                                                                     |             ------------------- cosphi 1.0      =   0.0 V = 12.0 mA
                                                                     |             underexcited        cosphi 0.95cap. =  -0.5 V = 10.6 mA
                                                                     |                                 cosphi 0.9 cap. =  -1.0 V =  9.3 mA
                                                                     |                                 cosphi 0.0 cap. = -10.0 V
                                                                     |  +------------+
                                                                     +--| scal. AO_mA|-------PF_AO_PF_I => AVR cosphi_setpoint 4/20mA
                                                                        +------------+

Outstandings:
------------
(*******************************************************************************)
PROGRAM _CYCLIC

// bestand:
	(* MMU values:     Werte von -0.0 .. -0.999 (untererregt) und 1.000 .. 0.00 (uebererregt) zulässig *) (* = 0,0 cap. .. 1 .. 0,0 ind. MMU values   *)
	(* PF lineariezed: Werte von  2.0 ..  1.001 (untererregt) und 1.000 .. 0.00 (uebererregt) zulässig *) (* = 0,0 cap. .. 1 .. 0,0 ind. LINEARISIERT *)

	(* linearization typical values *)
	(*  MMU    .. PF_lin .. PF                    *)
	(*  0.0    .. 0.0    .. 0.0  uebererregt(ind) *)
	(*  0.8    .. 0.8    .. 0.8  uebererregt(ind) *)
	(*  1.0    .. 1.0    .. 1.0                   *)
	(* -0.95   .. 1.05   .. 0,95 untererregt(cap) *)
	(*  0.0    .. 2.00   .. 0,0  untererregt(cap) *)

	(* ================================================================================================== *)
	(* linearisierung *)
	(*   y    .. PF_lin .. PF                   *)
	(*   0 %  .. 2.00   .. 0,0 untererregt(cap) *)
	(*  45 %  .. 1.10   .. 0,9 untererregt(cap) *)
	(*  50 %  .. 1.00   .. 1,0                  *)
	(*  80 %  .. 0.80   .. 0,8 uebererregt(ind) *)
	(* 100 %  .. 0.0    .. 0,0 uebererregt(ind) *)

	(* setting für mA or V -output *)
	(* mA for controller type BASLER DM110, NEWAGE RCI, AVK QPF *)	(* PF-Range mA Standard: -0,7 .. +0,7 =  4-20mA     *)
	(*  V for controller type BASLER DECS 100, ABB Unitrol,.... *)	(* PF-Range  V Standard: -0,7 .. +0,7 = -3V ... +3V *)
	(* ================================================================================================== *)

	(* P-limit for PF-controller with fixed values *) (* e.g. setpoint for cosphi 0,8 after sy *)
	GW_P_pfctr_fix := 0.250;	(* %P_Nom *)
	HY_P_pfctr_fix := 0.050;	(* %P_Nom *)

	(* PF-value for fixed PF-controller *)
	PF_1_fix := 1.000;		(* cosphi 1,0 *)
	PF_2_fix := 0.800;		(* cosphi 0,8 *)

	(* value for range without PF-controller *)
	U_fix := 1.000;

	(* ================================================================================================== *)
	(* PF-controller y fixed values *)
	(* P-limit *)
	xGR_MIN_PF_STELL(In := IN_GC.rP_Act_Norm_Filt, Gw := GW_P_pfctr_fix, Hy := HY_P_pfctr_fix);
	bPF_CosPCtr_Hold := xGR_MIN_PF_STELL.Q;

	(* controller stati *)
	IF Para.bPF_CosPCtr_Ena (*AND Para.iPF_CosPCtr_Choice > 0*) THEN
		IF NOT OUT_GC.tPF_CosPCtr_Ena.Do THEN
			yBlock  := 0.0;							(* 0% Q für cosphi 1.0 settings for idle run/engine stop [U-BEREICH] *)
			bBlock  := TRUE;						(* ohne Rampe bei Block2 *)
		ELSIF bPF_CosPCtr_Hold AND IN_GC.bEng_Dem THEN
			yBlock  := 0.02;						(* fix 2% Q, lastrampe bis aktivierung Q-controller *)
			bBlock  := TRUE;        				(* ohne Rampe bei Block2 *)
		ELSIF bPF_CosPCtr_Hold AND NOT IN_GC.bEng_Dem THEN
			yBlock  := 0.0;							(* cosphi 1.0 settings for deloading for engine stop *)
			bBlock  := TRUE;
		ELSE
			yBlock  := 0.0;							(* Spare *)
			bBlock  := FALSE;						(* controller modus [PF_Bereich] *)
		END_IF;
	ELSE
			yBlock  := 0.0;							(* without PF controller [U-BEREICH] *)
			bBlock  := TRUE;						(* ohne Rampe bei Block2 *)
	END_IF;

	//	(* Rangierung auf Regler *)
	OUT_GC.rPF_CosPCtr_block := yBlock;
	OUT_GC.bPF_CosPCtr_block := bBlock;

	(*------------------------------------------------------------------------------------------------------*)
	(* summation                                                                                            *)
	(*------------------------------------------------------------------------------------------------------*)
	rQ_Set_Lim;		(* from pf_ctr *)
	tCtr_Q_Out.Y;	(* ctr op.point: y = -1,0..0..+1,0  = -100%Qnom..0..+100%Qnom  *)

	CASE Para.iQ_GrC_PointCtrl OF
	0:	rQ_Set_Sum := rQ_Set_Lim + tCtr_Q_Out.Y;(* customer signal *)
	1:	rQ_Set_Sum := rQ_Set_Lim + tCtr_Q_Out.Y;(* MMD1 generator *)
	2:	rQ_Set_Sum := rQ_Set_Lim + tCtr_Q_Out.Y;(* MMD2 mains *)
	3:	rQ_Set_Sum := rQ_Set_Lim;               (* direct control without controller *)
	ELSE
		rQ_Set_Sum := rQ_Set_Lim + tCtr_Q_Out.Y;
	END_CASE;

	(*------------------------------------------------------------------------------------------------------*)
	OUT_GC.tPF_CosPCtr_Ena.Do;	 		 (* release gen.controller *)
	MM2VIS.bSel_AVR_Set := OUT_GC.tPF_CosPCtr_Ena.Do AND NOT bBlock;

	(*------------------------------------------------------------------------------------------------------*)
	(* Q_Set selection depending on engine operation status *)
	IF MM2VIS.bSel_AVR_Set THEN	rQ_AVR_Set := rQ_Set_Sum;	                                (* controller value -> AVR *)
    ELSE                        rQ_AVR_Set := OUT_GC.rPF_CosPCtr_block + rU_Gen_Diff_Match; (* engine operation depending set value *)
	END_IF;

	rQ_AVR_Set := LIMIT(Para.rQ_UnderExc_Lim, rQ_AVR_Set, Para.rQ_OverExc_Lim);

	MM2VIS.rQ_AVR_Set_Norm := rQ_AVR_Set;//display15

	(*======================================================================================================*)
	(* calculation rPF_POC_Set from rQ_Set_Sum (P_Act related to S_Nom!) *)
	IF    bBlock                    THEN rPF_POC_Set := 1.0;//yBlock for PF control;
	ELSIF Para.iQ_GrC_PointCtrl = 2 THEN
		IF	Para.rS_Nom > 0            THEN rPF_POC_Set := COS(ATAN(rQ_Set_Sum /(IN_GC.tP_Act[2].Ai/Para.rS_Nom)));(* erg.ohne vorzeichen! *)
		END_IF;
		IF rQ_Set_Sum < 0.0			   THEN rPF_POC_Set := rPF_POC_Set * (-1);
		END_IF;
	ELSE  														(* 1 or 3(direct control: P_Act[1]) *)
		IF	Para.rS_Nom > 0            THEN rPF_POC_Set := COS(ATAN(rQ_Set_Sum /(IN_GC.tP_Act[1].Ai/Para.rS_Nom)));(* erg.ohne vorzeichen! *)
		END_IF;
		IF rQ_Set_Sum < 0.0			   THEN rPF_POC_Set := rPF_POC_Set * (-1);
		END_IF;
	END_IF;

	(* linearization rPF_POC_Act *)
	(* +0,7(ind/overexc.)..1,0..-0,7(cap/underexc.) ==> 0,70 .. 1,00 .. 1,30 *)
	IF rPF_POC_Set >= 0 THEN rPF_POC_Set_lin := rPF_POC_Set;
	ELSE					 rPF_POC_Set_lin := rPF_POC_Set + 2.000;
	END_IF;

	(*------------------------------------------------------------------------------------------------------*)
	(* Werte für mA Ausgang*)
	(* PF setpoint y = 0.0 to 1.0 to 2.0 = 0.0ind. to 1.0 to 0.0cap. *)
	(* calculation voltage value for PF_lin = 1.30 = cosphi 0.7cap =  4.0mA *)
	(* calculation voltage value for PF_lin = 1.10 = cosphi 0.9cap =  9.3mA *)
	(* calculation voltage value for PF_lin = 0.70 = cosphi 0.7ind = 20.0mA *)
	xSigScal_PF_I(X := rPF_POC_Set_lin, X1 := 1.30, Y1 := 4.0, X2 := 0.70 , Y2 := 20.0);

	(* Output current restricted between 9.3mA to 20mA this corresponds to *)
    (* Restricted output range based on checklist 9.3mA TO 20.0mA *)
	OUT_GC.tPF_AO_PF_I.Ao := LIMIT(9.3, xSigScal_PF_I.Y_SCAL + rU_Gen_Diff_Match_I, 20.0);

	(*------------------------------------------------------------------------------------------------------*)
	(* Werte für V Ausgang*)
	(* PF setpoint y = 0.0 to 1.0 to 2.0 = 0.0ind. to 1.0 to 0.0cap. *)
	(* calculation voltage value for PF_lin = 0.00 = cosphi 0.0cap = -10V *)
	(* calculation voltage value for PF_lin = 1.00 = cosphi 1.0    =   0V *)
	(* calculation voltage value for PF_lin = 2.00 = cosphi 0.0ind = +10V *)
	xSigScal_PF_U(X := rPF_POC_Set_lin, X1 := 0.000, Y1 := 10.0, X2 := 2.000 , Y2 := -10.0);

	(* Output voltage restricted between -1.0V to +3.0V  this corresponds to *)
 	(* Restricted output range based on checklist -0.5V TO +2.5V *)
	OUT_GC.tPF_AO_PF_U.Ao := LIMIT (-0.5, xSigScal_PF_U.Y_SCAL + rU_Gen_Diff_Match_U, 2.5);

	(*-------------------------------------------------------------------------------------------------------*)
	(* Q set to AVR *)
	(*-------------------------------------------------------------------------------------------------------*)
	(* controller output    y = -1,0..0..+1.0% = -100%..0..+100%Qnom = cosphi 0.0cap .. 1.0 .. 0.0ind. *)
	(* Output voltage:  -2.7V =  -27%Qnom = cosphi -0.95 untererregt *)
	(*                   0.0V =    0%Qnom = cosphi  1.00             *)
    (*                  +6.0V =   60%Qnom = cosphi +0.80 uebererregt *)
	OUT_GC.tQ_AVR_Set_U.Ao := rQ_AVR_Set * 10;

	(*----------------------------------------------------------------------------------*)
	Para.iQ_GrC_CtrlFun;		(* selection Q function  	                        	*)
	Para.iQ_GrC_PointCtrl;		(* selection point of control (POC)                    	*)
	Para.bPF_CosPCtr_Ena;		(* generator controller active                          *)

	OUT_GC.tPF_CosPCtr_Ena.Do;	(* demand cosphi from limit Pgen, gcb_on, mcb_on		*)
	OUT_GC.bPF_CosPCtr_block;	(* demand y_BLOCK2										*)
	OUT_GC.rPF_CosPCtr_block;	(* set value y_block 									*)
	OUT_GC.rPF_AO_PF_I;	        (* AO=mA: controller value to generator controller(AVR)	*)
	OUT_GC.rPF_AO_PF_U;	        (* AO=V:  controller value to generator controller(AVR) *)
	OUT_GC.tQ_AVR_Set_U.Ao;     (* AO=V:  Qset value to generator controller(AVR) 		*)
	(*----------------------------------------------------------------------------------*)

	(*-------------------------------------------------------------------------------------------------------*)
	(* generator air inlet temperature to generator controller - for UNITROL internal power limitation *)
	IF Para.bT_GenAirIn_Active AND Para.bT_GenAirIn2_Active THEN
		IF    MM2VIS.bMsg2555 AND MM2VIS.bMsg3468 THEN OUT_GC.tT_AO_Gen_T_In.Ao :=  0;
		ELSIF MM2VIS.bMsg2555                     THEN OUT_GC.tT_AO_Gen_T_In.Ao :=  IN_GC.tGen_T_In2.Ai;
		ELSIF MM2VIS.bMsg3468                     THEN OUT_GC.tT_AO_Gen_T_In.Ao :=  IN_GC.tGen_T_In.Ai;
		ELSE                                           OUT_GC.tT_AO_Gen_T_In.Ao := (IN_GC.tGen_T_In.Ai + IN_GC.tGen_T_In2.Ai)/2; (* average *)
		END_IF;
	ELSIF Para.bT_GenAirIn_Active THEN
		IF MM2VIS.bMsg2555 THEN OUT_GC.tT_AO_Gen_T_In.Ao := 0;
		ELSE					OUT_GC.tT_AO_Gen_T_In.Ao := IN_GC.tGen_T_In.Ai;
		END_IF;
	ELSE
		IF IN_GC.bAMM_T_Ch_T1LP_Avg  THEN 	OUT_GC.tT_AO_Gen_T_In.Ao := 0;
		ELSE							    OUT_GC.tT_AO_Gen_T_In.Ao := IN_GC.rT_Ch_T1LP_Avg;
		END_IF;
	END_IF;

	(* power reduction according high generator air in temperature *)
	IF Para.bT_GenAirIn_Active OR Para.bT_GenAirIn2_Active THEN
		IF MM2VIS.bMsg2555 AND MM2VIS.bMsg3468 THEN
			OUT_GC.rP_Red_T_GenAirIn_Norm := 1;
		ELSE
			OUT_GC.rP_Red_T_GenAirIn_Norm := LIMIT(0.5, (1 - ((OUT_GC.tT_AO_Gen_T_In.Ao - Para.rT_Pred_GenAirIn_Start) * Para.rT_Pred_GenAirIn_Rate)), 1.0);
		END_IF;
	ELSE
		OUT_GC.rP_Red_T_GenAirIn_Norm := 1;
	END_IF;

	(*-------------------------------------------------------------------------------*)
	(* Release for Unitrol *)
	OUT_GC.tGCB_On_ReturnSign.Do := IN_GC.tGCB_On.Di;

	(*------------------------------------------------------------------*)
END_PROGRAM
```

#### pf_custInit.st
```iecst
(*********************************************************************
pf_cust  Initialization

This code is confidential and proprietary to the INNIO Company.
It may not be used in any form, or reproduced in any manner,
without the express written permission of the INNIO Company.
Copyright, INNIO Company, 2019

Customized modifications: -
------------------------

History:
-------

 ********************************************************************)

PROGRAM _INIT

END_PROGRAM
```

#### pf_cust.var
```iecst
VAR
	bPF_CosPCtr_Hold : BOOL; (*Q controller on hold*)
	bBlock : BOOL;
	GW_P_pfctr_fix : REAL;
	HY_P_pfctr_fix : REAL;
	xGR_MIN_PF_STELL : GR_MINR;
	yBlock : REAL;
	rQ_AVR_Set : REAL; (*Q setpoint to AVR [%]*)
	xSigScal_PF_I : xSigScal_R; (*scaling mA output *)
	xSigScal_PF_U : xSigScal_R; (*scaling V output *)
	rPF_POC_Set : REAL;
	rPF_POC_Set_lin : REAL;
END_VAR
```

### Program Logical/Generator/v_ctr (IEC, version 4.13.0) - voltage control

#### v_ctrCyclic.st
```iecst
	(*******************************************************************************
	v_ctr		voltage control and matching for synchronisation (cyclic)
				Offset signal for dig. generator controller for voltage matching

	This code is confidential and proprietary to the INNIO Company.
	It may not be used in any form, or reproduced in any manner, without the express
	written permission of the INNIO Company.
	Copyright, INNIO Company, 2021

	Customized modifications: -
	------------------------

	History:
	-------
	V0.10	16-07-2007	Wasserer, 	generated
	V3.20.0	11.11.2010	lettenb. 	v_match included into v_ctr for standardization
			07.12.2010	lettenb.	u_adj_speed_a  	:= FALSE = default
	V3.30.0	28.10.2011	Tinello		parameter "nominal frequency" was increased by factor 10
			22.11.2011	Wasserer, 	Auswahl SY mit externe +/- Befehle oder über MMU Berechnung eingefügt
	V4.00.1 21.05.2014	lettenb.	scaling to V, mA changed, cleanup
	V4.00.2 27.05.2014	lettenb.	workaround, definition of new parameters
			02.07.2014				xSigScal_uoffset_f: Y1:= -0.10, Y2:= 0.10 setted, bugfix
	V4.00.3 29.07.2014				IN_GC.tU_DI_Gen_Inc.Di,IN_GC.tU_DI_Gen_Dec.Di removed(war mit einführung xt4 doppelt angelegt)
	V4.00.4 29.07.2014				bU_plus_MMU,bU_minus_MMU: Eng_Run added(relais taktet ständig bei motorstillstand)(cornee)
	V4.00.5 28.01.2015				voltage adjustment from pb8 included
	V4.03.0 03.08.2015	lettenb.	LIMIT(Para.rU_adj_max_down: -vorzeichen entfernt, bugfix(kirchler peter)
	V4.04.0 31.10.2016				xSigScal_u_offset_V.X1/2, xSigScal_u_offset_mA.X1/2	corr., bugfix(wasserer/rosenheim)
	V4.05.0 13.12.2017				rU_Gen_Diff_Match added for Ctr_Q, write parameter removed(code guide line)
	V4.05.7 10.10.2018	lettenb.	voltage matching puls duration depending on voltage differenz(kirchmair)
			19.12.2018	Hohensinner	added voltage droop and offset for island mode
	V4.07.0	03.04.2019	Hohensinner replaced voltage set point with actual voltage on HMI working point
	V4.07.1	03.06.2019	Hohensinner deactivated generator controller reset if in droop mode or external voltage setpoint active
	V4.09.0 06.08.2019	lettenb.	OUT_GC.tGenCtrResetSp.Do: IN_GC.tGCB_DVM.Di added, reset unitrol for RSY voltage matching with MSY, bugfix
	V4.11.0 29.09.2021	lettenb.	release voltage control by customer bit IN_GC.bN_U_Set_Ext_On added, bugfix
			11.10.2021	Hohensinner	added reactive power setpoint for voltage droop mode
			21.01.2022	MayerR      External voltage and reactive power for droop mode setpoint with corresponding parameter selection added
	V4.13.0 07.03.2024	Farre,		issue #890, #1089: delete scaling analog input signals and shifted to HalIO

	Instructions for use:
	--------------------

	Outstandings:
	------------

    Description:
    ==================================================================
    Matching the generator voltage by the analog signal (Offset-Signal) to the digital Generator controller
	Additional offset in "voltage regulated operation:

    Voltage Adjustment:
	Nominal voltage generator from multi measurement unit - PAR
    Generator voltage - Setpoint at 0% PN from PAR
    Generator voltage - Setpoint at 100% PN aus PAR
    Factor for Voltage adjustment speed from PAR
    Maximum Adjustment range (+/- 10%) from PAR

	- during SY Voltage setpoint is increased/decreased
	- Deviation of the Voltage setpoint from nominal voltage is Uoffset
    - Limit the deviation according to the maximum adjustment range
	- Re-calculate the Uoffset to units of the device (mV or mA)

	Beschreibung:
	===================================================================
	Anpassung der Generatorspannung mithilfe des Analogsignals (Offset-Signal) an den dig. Generatorregler
	Verwendung des Signales aus pf_ctr, pf_cust (diane cos-phi-controller)
	zusätzlicher Offset im "spannungsgeregelten Betrieb"

	Spannungsverstellung:
	Nennspannung Generator aus Multimessumformer-PAR
	Soll-Generatorspannung bei 0% PN aus PAR
	Soll-Generatorspannung bei 100% PN aus PAR
	Faktor für Spannungsverstellgeschwindigkeit aus PAR
	max. Verstellbereich ( +/- 10% ) aus PAR

	- während SY wird die Sollspannung erhöht/verringert
	- Abweichung der Sollspannung zur Nennspannung entspricht dem Uoffset
	- Limitierung der Abweichung gemäß max. Verstellbereich
	- Umrechnung des Uoffset auf Einheiten der Karte (in mV oder mA)

	Impulsdauer: Anpassung an die Spannungsabweichung, je größer die Abweichung desto länger der Impuls.
	Maximalwert ist 1500ms was 1,5% entspricht, Minimalwert 150ms was 0,15% entsprich.
	Dadurch hat der Unitrol dann noch 500ms um sich auszuregeln, bevor wir den nächsten Takt freigaben.
	Je weiter wir uns dem Sollwert nähern, desto kürzer wird dann der Impuls.(kirchmair)

	*********************************************************************************)
PROGRAM _CYCLIC

	IF IN_GC.bN_U_Set_Ext_On THEN		(*release voltage control by customer bit(AB energy)*)
		iSrc_U_OffsSet := 2;
	ELSE
		iSrc_U_OffsSet := Para.iSource_U_OffsSet;
	END_IF;
	MM2VIS.iSource_U_OffsSet := iSrc_U_OffsSet;

	(* generator voltage adjustment from Di *)
	OUT_GC.tU_MidPos.Do :=	NOT IN_GC.bGCB_DemSy
						AND NOT IN_GC.bMCB_DemSy
						AND NOT IN_GC.tGCB_DVM.Di
						AND 	Para.bSyActive;

	OUT_GC.tU_Plus.Do :=   (IN_GC.bGCB_DemSy OR IN_GC.bMCB_DemSy OR IN_GC.tGCB_DVM.Di OR NOT Para.bSyActive)
						AND(bU_plus_MMU OR IN_GC.tU_Adj_Plus.Di);

	OUT_GC.tU_Minus.Do:=   (IN_GC.bGCB_DemSy OR IN_GC.bMCB_DemSy OR IN_GC.tGCB_DVM.Di OR NOT Para.bSyActive)
						AND(bU_minus_MMU OR IN_GC.tU_Adj_Minus.Di);

	(* generator controller reset set point (UNITROL), reset voltage offset for island operation *)
	OUT_GC.tGenCtrResetSp.Do :=	IN_GC.tGCB_On.Di
						AND NOT IN_GC.tGCB_DVM.Di 				(* reset unitrol for RSY voltage matching *)
						AND     IN_GC.tEng_Run.Do
						AND NOT IN_GC.tMCB_On.Di
						AND NOT IN_GC.bMCB_DemSy
						AND NOT OUT_GC.tPF_CosPCtr_Ena.Do
						AND iSrc_U_OffsSet = 0;		(* disable, if in droop mode or external setpoint active *)

	(* ============================================================================= *)
	(* ============================================================================= *)
	(* Scaling external U - Setpoint (Island operation) - Hardware*)
	IF (Para.iU_Isl_SetX = 5) THEN
		(* Generierung Messsignalstörung *)
		IF Para.rU_SetExtAI_SetI1 >= 4.0 AND Para.rU_SetExtAI_SetI2 >= 4.0 AND IN_GC.tU_SetExtAI_Norm.GoodQual AND Para.bRelFreeze_Uset_Isl THEN
			rBuffer_U_SetExt[x_U_SetExt] := IN_GC.tU_SetExtAI_Norm.Ai;
			x_U_SetExt := x_U_SetExt + 1;
			IF x_U_SetExt > 9 THEN
				x_U_SetExt := 0;
				bBuffer_U_SetExt := TRUE;
			END_IF;
		END_IF;

		IF NOT bBuffer_U_SetExt THEN
			rLCRLimScal_U_SetExt_old := 0.00;
		END_IF;

		xTON_GoodQual_U_SetExt(IN := IN_GC.tU_SetExtAI_Norm.GoodQual, PT := tiGoodQual);

		IF Para.rU_SetExtAI_SetI1 >= 4.0 AND Para.rU_SetExtAI_SetI2 >= 4.0 AND NOT xTON_GoodQual_U_SetExt.Q THEN
			bMsg9285 := TRUE;
			IF Para.bRelFreeze_Uset_Isl AND bBuffer_U_SetExt  THEN
				rU_setExt := rLCRLimScal_U_SetExt_old;
			END_IF;
		ELSE
			bMsg9285 := FALSE;
			rU_setExt := IN_GC.tU_SetExtAI_Norm.Ai;

			IF Para.bRelFreeze_Uset_Isl THEN
				z_U_SetExt := x_U_SetExt - 8;
				IF bBuffer_U_SetExt THEN
					IF z_U_SetExt >= 0 THEN
						rLCRLimScal_U_SetExt_old := rBuffer_U_SetExt[z_U_SetExt];
					ELSE
						rLCRLimScal_U_SetExt_old := rBuffer_U_SetExt[z_U_SetExt + 9];
					END_IF;
				ELSE
					rLCRLimScal_U_SetExt_old := 0.00;
				END_IF;
			END_IF;
		END_IF;

	ELSE
		rU_setExt := 0.00;
		bMsg9285  := FALSE;
	END_IF;

	(**********************************************************)
	(* Selection of external U - Setpoint (Island operation)  *)
	(**********************************************************)
	rUset_Isl := 0.0;
	bUset_Isl := FALSE;

	(* Choice for reactive power functions *)
	CASE Para.iU_Isl_SetX OF
	0:  (* NOT USED *)
		bUset_Isl := FALSE;
	1:  (* INTERN *)
		rUset_Isl := Para.rU_Isl_SetInt;
		bUset_Isl := TRUE;
	2:  (* EXTERN DI - spare *)
		rUset_Isl := Para.rU_Isl_SetAct_BU;
		bUset_Isl := FALSE;
	3:  (* EXTERN BUS *)
		IF (Para.bComm1_Ena OR Para.bComm2_Ena) AND NOT IN_GC.bMsg1147 THEN	(* Bus active and without communication failure *)
			rUset_Isl := IN_GC.rUset_Isl_Bus;
		ELSE
			rUset_Isl := Para.rU_Isl_SetAct_BU;
		END_IF;
		bUset_Isl := TRUE;
	4:  (* CUSTOM - prepared for project specific use *)
		IF TRUE THEN
			rUset_Isl := IN_GC.rU_Set_Norm_Cust;
		ELSE
			rUset_Isl := Para.rU_Isl_SetAct_BU;
		END_IF;
		bUset_Isl := TRUE;
	5:  (* EXTERN AI *)
		IF IN_GC.bExtCtrOk THEN (* External input is able to be read if external activations or HMI activation *)
			IF NOT bMsg9285 OR Para.bRelFreeze_Uset_Isl THEN
				rUset_Isl := rU_setExt;
			ELSE
				rUset_Isl := Para.rU_Isl_SetAct_BU;
			END_IF;
		ELSE
			rUset_Isl := Para.rU_Isl_SetAct_BU;
		END_IF;
		bUset_Isl := TRUE;
	ELSE
		bUset_Isl := FALSE;
	END_CASE;

	(**********************************************************)
	(* RESULTS - External U - Setpoint (Island operation) 	  *)
	(**********************************************************)
	rUset_Isl;
	bUset_Isl;

	(* ============================================================================= *)
	(* Scaling external reactive power setpoint for frequency droop mode - Hardware*)
	IF (Para.iQ_Droop_SetX = 5) THEN
		(* Generierung Messsignalstörung *)
		IF Para.rQ_Droop_Set_SetI1 >= 4.0 AND Para.rQ_Droop_Set_SetI2 >= 4.0 AND IN_GC.tQ_Droop_Set.GoodQual AND Para.bRelFreeze_Qset_Droop THEN
			rBuffer_Q_Droop_Set[x_Q_Droop_Set] := IN_GC.tQ_Droop_Set.Ai;
			x_Q_Droop_Set := x_Q_Droop_Set + 1;
			IF x_Q_Droop_Set > 9 THEN
				x_Q_Droop_Set := 0;
				bBuffer_Q_Droop_Set := TRUE;
			END_IF;
		END_IF;

		IF NOT bBuffer_Q_Droop_Set THEN
			rLCRLimScal_Q_Droop_Set_old := 0.00;
		END_IF;

		xTON_GoodQual_Q_Droop_Set(IN := IN_GC.tQ_Droop_Set.GoodQual, PT := tiGoodQual);

		IF Para.rQ_Droop_Set_SetI1 >= 4.0 AND Para.rQ_Droop_Set_SetI2 >= 4.0 AND NOT xTON_GoodQual_Q_Droop_Set.Q THEN
			bMsg9351 := TRUE;
			IF Para.bRelFreeze_Qset_Droop AND bBuffer_Q_Droop_Set  THEN
				rQset_Droop := rLCRLimScal_Q_Droop_Set_old;
			END_IF;
		ELSE
			bMsg9351 := FALSE;
			rQ_Droop_SetExt	:= IN_GC.tQ_Droop_Set.Ai;

			IF Para.bRelFreeze_Qset_Droop THEN
				z_Q_Droop_Set := x_Q_Droop_Set - 8;
				IF bBuffer_Q_Droop_Set THEN
					IF z_Q_Droop_Set >= 0 THEN
						rLCRLimScal_Q_Droop_Set_old := rBuffer_Q_Droop_Set[z_Q_Droop_Set];
					ELSE
						rLCRLimScal_Q_Droop_Set_old := rBuffer_Q_Droop_Set[z_Q_Droop_Set + 9];
					END_IF;
				ELSE
					rLCRLimScal_Q_Droop_Set_old := 0.00;
				END_IF;
			END_IF;
		END_IF;

	ELSE
		rQ_Droop_SetExt	:= 0.00;
		bMsg9351		:= FALSE;
	END_IF;

	(***************************************************************************)
	(* Selection of external reactive power setpoint for frequency droop mode  *)
	(***************************************************************************)
	rQset_Droop	:= 0.0;
	bQset_Droop	:= FALSE;

	(* Choice for reactive power functions *)
	CASE Para.iQ_Droop_SetX OF
	0:  (* NOT USED *)
		bQset_Droop	:= FALSE;
		MM2VIS.iIdx_Q_Droop_Offs := 0;
	1:  (* INTERN *)
		rQset_Droop	:= Para.rQ_Droop_SetInt / MAX(1, Para.rS_Nom);
		bQset_Droop	:= TRUE;
	2:  (* EXTERN DI - spare *)
		rQset_Droop	:= Para.rQ_Droop_SetAct_BU / MAX(1, Para.rS_Nom);
		bQset_Droop	:= FALSE;
	3:  (* EXTERN BUS *)
		IF (Para.bComm1_Ena OR Para.bComm2_Ena) AND NOT IN_GC.bMsg1147 THEN (* Bus active and without communication failure *)
			rQset_Droop	:= IN_GC.rQset_Droop_Bus;
		ELSE
			rQset_Droop	:= Para.rQ_Droop_SetAct_BU / MAX(1, Para.rS_Nom);
		END_IF;
		bQset_Droop	:= TRUE;
		MM2VIS.iIdx_Q_Droop_Offs := 2;
	4:  (* CUSTOM - prepared for project specific use *)
		IF TRUE THEN
			rQset_Droop; // := Connectanything;
		ELSE
			rQset_Droop := Para.rQ_Droop_SetAct_BU / MAX(1, Para.rS_Nom);
		END_IF;
		bQset_Droop	:= TRUE;
	5:  (* EXTERN AI *)
		IF IN_GC.bExtCtrOk THEN (* External input is able to be read if external activations or HMI activation *)
			IF NOT bMsg9351 OR Para.bRelFreeze_Qset_Droop THEN
				rQset_Droop	:= rQ_Droop_SetExt;
			ELSE
				rQset_Droop	:= Para.rQ_Droop_SetAct_BU / MAX(1, Para.rS_Nom);
			END_IF;
		ELSE
			rQset_Droop	:= Para.rQ_Droop_SetAct_BU / MAX(1, Para.rS_Nom);
		END_IF;
		bQset_Droop	:= TRUE;
		MM2VIS.iIdx_Q_Droop_Offs := 1;
	ELSE
		bQset_Droop	:= FALSE;
	END_CASE;

	(******************************)
	(* RESULTS - External reactive power setpoint for frequency droop mode 	  *)
	(******************************)
	rQset_Droop;
	bQset_Droop;

	(* ============================================================================= *)
	(* voltage controller *)

	(* generate rate signal for voltage adjustment*)
	xTON_U_TAKT(IN := NOT xTON_U_TAKT.Q, PT := T#2s);
	xTON_U_TAKT_P(IN := xTON_U_TAKT.Q, PT := T#500ms);
	U_TAKT := xTON_U_TAKT.Q;

	(* MMU Synch 1 *)
	(* ============================================================================= *)
	(* controller deadband 0,5% and voltage difference*)
	IF NOT IN_GC.bSyncSlipMode[2] THEN
		rU_SY_span := 0.005 * Para.rU_SyncNom[1];
		rU_SY_diff := IN_GC.tU_MMD_Synch2[1].Ai - IN_GC.tU_MMD_Synch1[1].Ai;
	ELSE
		rU_SY_span := 0.005 * Para.rU_SyncNom[2];
		rU_SY_diff := IN_GC.tU_MMD_Synch2[1].Ai - IN_GC.tU_MMD_Synch1[2].Ai;
	END_IF;

	(* pulse duration depending on voltage difference *)
	IF Para.rU_SyncNom[1] > 0 THEN											(*avoid division by zero*)
		rU_diff_percent := ABS(rU_SY_diff / Para.rU_SyncNom[1] * 100);		(*voltage difference in %*)
		tiPuls := (REAL_TO_TIME(LIMIT(150, rU_diff_percent * 1000, 1500)));	(*calc.pulse duration, min=150ms/max=1500ms*)
	END_IF;

	(* negative deviation => generator voltage to high *)
	bU_SyD_Dec := (rU_SY_diff < 0) AND (ABS(rU_SY_diff) > rU_SY_span);

	(* positive deviation => generator voltage to low *)
	bU_SyD_Inc := (rU_SY_diff > 0) AND (ABS(rU_SY_diff) > rU_SY_span);

	(* voltage adjustment down *)
	xTP_U_DOWN(IN:= bU_SyD_Dec AND EDGEPOS(U_TAKT), PT := tiPuls);
	bU_minus_MMU := IN_GC.tEng_Run.Do AND xTP_U_DOWN.Q;

	(* voltage adjustment up *)
	xTP_U_UP  (IN:= bU_SyD_Inc AND EDGEPOS(U_TAKT), PT := tiPuls);
	bU_plus_MMU	 := IN_GC.tEng_Run.Do AND xTP_U_UP.Q;

	(* voltage matching *)
	(* ============================================================================= *)
	(* Eingangskopplung *)
	(* ============================================================================= *)
	IN_GC.tU_Gen_Dec.Di;			(* Verstellbefehl -U von extern *) 		(* adjustment command -U External *)
	IN_GC.tU_Gen_Inc.Di;			(* Verstellbefehl +U von extern *)		(* adjustment command +U External *)

	Para.rU_Gen_Nom[1];				(* Nennspannung *)						(* nominal voltage *)
	Para.rF_Nom[1];					(* Nennfrequenz *)						(* nominal frequency *)
	IN_GC.tF_MMD[1].Ai;				(* IST-Frequenz *)						(* actual frequency *)

	(* Parameteranbindung *)
	Para.bU_Gen_Mns_Match;			(* Funktion Voltage matching über Analogsignal aktiv *)		(* Function voltage matching using analog signal active *)
	Para.rU_adj_max_up;		 		(* max.Verstellbereich Generatorspannung nach oben  +10% *)	(* max.adjustment generator voltage up   *)
	Para.rU_adj_max_down;		 	(* max.Verstellbereich Generatorspannung nach unten -10% *)	(* max.adjustment generator voltage down *)

	Para.rU_Gen_Rmp_Inc;		 	(* Rampe Spannungsverstellung %Un/s nach oben  +10% *)		(* max.adjustment generator voltage up   *)
	Para.rU_Gen_Rmp_Dec;		 	(* Rampe Spannungsverstellung %Un/s nach unten -10% *)		(* max.adjustment generator voltage down *)

	Para.rU_Gen_Diff_Idle;			(* U Offset im Leerlauf,   % UN *) 							(* U Offset in idle,      % UN *)
	Para.rU_Gen_Diff_Pn;			(* U Offset bei 100% Last, % UN *) 							(* U offset at 100% Load, % UN *)
									(* Vorbereitung für Inselbetrieb *)

	(* ex settings *)
	Para.bU_adj_gcb_mmd_calc_a;		(* U-verstellung synch.GCB mit MMU-Berechung aktiv *)
	Para.bU_adj_mcb_mmd_calc_a;		(* U-verstellung synch.MCB mit MMU-Berechung aktiv *)

	Para.bU_adj_gcb_ext_hilo_a;		(* U-verstellung synch.GCB mit externen höher/tiefer Verstellbefehlen aktiv *)
	Para.bU_adj_mcb_ext_hilo_a;		(* U-verstellung synch.MCB mit externen höher/tiefer Verstellbefehlen aktiv *)

	Para.bU_Gen_spd_match;			(* U-verstellung drehzahlabhängig aktiv - Spannungsknie im Inselbetrieb *)	(* U-adjustment speed dependent active - Voltage knee in Island operation *)
	Para.bU_Gen_P_Ena;				(* U-verstellung leistungsabhängig aktiv - "Statik" im Inselbetrieb *)		(* U-adjustment power dependent active - "Static" in Island mode *)
	Para.rU_Gen_match_delta;		(* U-verstellung pro Impuls z.B. 5 Promille UN / s *)						(* U-voltage per impulse e.g. 5 ppm UN/s *)
 	(* ============================================================================= *)

	Para.rF_Gen_Match_Min;			(* max.Verstellbereich Generatorfrequenz nach unten 5% *)	(* max.adjustment generator voltage up *)
	Para.rF_Gen_Match_Max;			(* max.Verstellbereich Generatorfrequenz nach oben  5% *)	(* max.adjustment generator voltage up *)
	(* ============================================================================= *)

	OUT_GC.bU_SyD_match :=	IN_GC.tEng_Run.Do		(* Anforderung Spannungsverstellung während SY *)	(* Demand Voltage adjustment during SY *)
					AND	NOT xOpMode.NetP
					AND    (IN_GC.tGCB_DVM.Di OR IN_GC.bGen_SyD_Dem);

	IF Para.bU_Gen_Mns_Match THEN
		(* ============================================================================= *)
		(* Spannungverstellung *)		(* Voltage adjustment *)
		(* ============================================================================= *)

		u_plus 		:= (IN_GC.bGCB_DemSy  AND Para.bU_adj_gcb_mmd_calc_a AND bU_plus_MMU)
					OR (IN_GC.bGCB_DemSy  AND Para.bU_adj_gcb_ext_hilo_a AND IN_GC.tU_Gen_Inc.Di)
					OR (IN_GC.bMCB_DemSy  AND Para.bU_adj_mcb_mmd_calc_a AND bU_plus_MMU)
					OR (IN_GC.tGCB_DVM.Di AND Para.bU_adj_mcb_ext_hilo_a AND IN_GC.tU_Gen_Inc.Di);

		u_minus 	:= (IN_GC.bGCB_DemSy  AND Para.bU_adj_gcb_mmd_calc_a AND bU_minus_MMU)
					OR (IN_GC.bGCB_DemSy  AND Para.bU_adj_gcb_ext_hilo_a AND IN_GC.tU_Gen_Dec.Di)
					OR (IN_GC.bMCB_DemSy  AND Para.bU_adj_mcb_mmd_calc_a AND bU_minus_MMU)
					OR (IN_GC.tGCB_DVM.Di AND Para.bU_adj_mcb_ext_hilo_a AND IN_GC.tU_Gen_Dec.Di);

		(* SY + Beruhigungszeit nach dem zuschalten *)(* SY + Relaxation time after switching ON *)
		xTOF_Synch(IN := OUT_GC.bU_SyD_match, PT := T#5s);

		(* Spannungsverstellung während SY *)(* Voltage adjustment during synchronization *)
		xR_TRIG_u_plus (CLK := u_plus);
		xR_TRIG_u_minus(CLK := u_minus);
		IF xTOF_Synch.Q THEN
			IF xR_TRIG_u_plus.Q THEN
				rU_Gen_Diff_Match_sy := rU_Gen_Diff_Match_sy + Para.rU_Gen_match_delta;
			END_IF;
			IF xR_TRIG_u_minus.Q THEN
				rU_Gen_Diff_Match_sy := rU_Gen_Diff_Match_sy - Para.rU_Gen_match_delta;
			END_IF;
		ELSE
			rU_Gen_Diff_Match_sy := 0.0;	(* "Return"-Funktion *)
		END_IF;

		rU_Gen_Diff_Match_sy :=  LIMIT(2 * Para.rU_adj_max_down, rU_Gen_Diff_Match_sy, 2 * Para.rU_adj_max_up);	(* Limitierung *)
		xRAMPE_rU_Gen_Diff_Match_sy(enable:= IN_GC.bEng_Dem OR M_HDREHZ, In:= rU_Gen_Diff_Match_sy, Rise:= Para.rU_Gen_Rmp_Inc, Sink:= Para.rU_Gen_Rmp_Dec, TC_Time:= 100);
	    rU_Gen_sy_match := xRAMPE_rU_Gen_Diff_Match_sy.Out;

		(* Spannungsverstellung leistungsabhängig - "Statik" im Inselbetrieb *)(* Voltage adjustment power dependent - "Static" in Island mode operation *)
		bU_Gen_P_match :=  Para.bU_Gen_P_Ena AND xOpMode.Island;
		IF bU_Gen_P_match THEN
			xSigScal_uoffset_p(X:= IN_GC.rP_Act_Norm_Filt, X1:= 0.000, Y1:= LIMIT(Para.rU_adj_max_down, Para.rU_Gen_Diff_Idle, Para.rU_adj_max_up),
			                                               X2:= 1.000, Y2:= LIMIT(Para.rU_adj_max_down, Para.rU_Gen_Diff_Pn,   Para.rU_adj_max_up));
			rU_Gen_Diff_Match_p := xSigScal_uoffset_p.Y_SCAL;
		ELSE
			rU_Gen_Diff_Match_p := 0;
		END_IF;
		rU_Gen_Diff_Match_p := LIMIT(2 * Para.rU_adj_max_down, rU_Gen_Diff_Match_p, 2 * Para.rU_adj_max_up);		(* Limitierung *)
		xRAMPE_rU_Gen_Diff_Match_p(enable:= IN_GC.bEng_Dem OR M_HDREHZ, In:= rU_Gen_Diff_Match_p, Rise:= Para.rU_Gen_Rmp_Inc, Sink:= Para.rU_Gen_Rmp_Dec, TC_Time:= 100);
		rU_Gen_P_match := xRAMPE_rU_Gen_Diff_Match_p.Out;

		(* Spannungsverstellung drehzahlabhängig - Spannungsknie im Inselbetrieb *)
		(* Voltage adjustment speed dependent - Voltage knee in Island mode operation *)
		OUT_GC.bU_Gen_match_isolated := Para.bU_Gen_spd_match
		                      	AND		xOpMode.Island
		                        AND    (IN_GC.rP_Act_Norm_Filt > 0.10) 	(* Werte für Freigabe bei Leistungsgrenze xx anpassen ! *)
		                        AND	NOT	IN_GC.tGen_Exc_Off.Di;

		IF OUT_GC.bU_Gen_match_isolated THEN
			IF Para.rF_Nom[1] > 0 THEN
				rF_Act_norm := IN_GC.tF_MMD[1].Ai / Para.rF_Nom[1];
			END_IF;
			xSigScal_uoffset_f(X:= rF_Act_norm, X1:= Para.rF_Gen_Match_Min, Y1:= -0.10, X2:= Para.rF_Gen_Match_Max, Y2:= 0.10);   (* Werte für Skalierung anpassen : 5% f-Abweichung -> 10% U-Abweichung *)
			u_offset_f := xSigScal_uoffset_f.Y_SCAL;
		ELSE
			u_offset_f := 0.0;
		END_IF;

		u_offset_f := LIMIT(2 * Para.rU_adj_max_down , u_offset_f, 2 * Para.rU_adj_max_up );		(* Limitierung *)
		xRAMPE_u_offset_f(enable := FALSE, In:= u_offset_f, Rise:= Para.rU_Gen_Rmp_Inc, Sink:= Para.rU_Gen_Rmp_Dec, TC_Time:= 100);	//rampe nicht aktiv
		rU_Gen_f_match := xRAMPE_u_offset_f.Out;

		(* neuer Spannungs-Offset*)
		(* New Voltage - Offset *)
		u_offset := rU_Gen_P_match + rU_Gen_sy_match + rU_Gen_f_match;
		u_offset := LIMIT(Para.rU_adj_max_down , u_offset, Para.rU_adj_max_up);			(* Limitierung der gesamten Spannungsverstellung *)

		rU_Gen_Diff_Match := u_offset;

		(* Scaling for mA
		   Basler DM110: Voltage regulation 4-20mA = -15% to +15% Usetpoint
		   Normal Setpoint => 12mA
		   ==> Offset-Signal: -8mA to +8mA = -15% to +15% *)
		xSigScal_u_offset_mA.X  := u_offset;
		xSigScal_u_offset_mA.X1 := -0.15;
		xSigScal_u_offset_mA.X2 := +0.15;
		xSigScal_u_offset_mA.Y1 := -8.0;		(* -8mA *)
		xSigScal_u_offset_mA.Y2 := +8.0;		(* +8mA *)
		xSigScal_u_offset_mA();

		rU_Gen_Diff_Match_I := xSigScal_u_offset_mA.Y_SCAL;			(* Ausgangssignal siehe task: pf_cust *)

		(* Scaling for V
		   Basler DEC100: Voltage regulation -3V to +3V = -30% to +30% Usetpoint
		   Normal Setpoint => 0V
		   ==> Offset-Signal: -3V to +3V = -30% to +30%	*)
		xSigScal_u_offset_V.X  := u_offset;
		xSigScal_u_offset_V.X1 := -0.30;
		xSigScal_u_offset_V.X2 := +0.30;
		xSigScal_u_offset_V.Y1 := -3.0;			(* -3V *)
		xSigScal_u_offset_V.Y2 := +3.0;			(* +3V *)
		xSigScal_u_offset_V();

		rU_Gen_Diff_Match_U  := xSigScal_u_offset_V.Y_SCAL;	(* Ausgangssignal siehe task: pf_cust *)
													        (* Output signal see task: pf_cust *)

	ELSE
		rU_Gen_Diff_Match_I := 0;
		rU_Gen_Diff_Match_U := 0;
		rU_Gen_Diff_Match   := 0;
	END_IF;

	(** U: Voltage static *)

	(** U.1.0: calculate rQ_Nom *)
	IF Para.rEta_Gen_PF08 <> 0 AND Para.rEta_Gen_PF1 <> 0 THEN
		rP_Nom_PF08	:= IN_GC.rP_Nom / Para.rEta_Gen_PF1 * Para.rEta_Gen_PF08;
	ELSE
		rP_Nom_PF08	:= IN_GC.rP_Nom;
	END_IF;
	IF (Para.rS_Nom ** 2) - (rP_Nom_PF08 ** 2) > 0 THEN
		rQ_Nom := ((Para.rS_Nom ** 2) - (rP_Nom_PF08 ** 2))**(0.5);
	ELSE
		rQ_Nom := 0.0;
	END_IF;

	(** U.1.3: set source and visualization *)
	IF VIS2MM.bQ_Droop_Set_Man THEN			(* Droop Offset manual via HMI *)
		rQ_Offs_Input := VIS2MM.rQ_Droop_Set_Man;
		MM2VIS.iIdx_Q_Droop_Offs := 3;
	ELSE 									(* Droop Offset from other sources - see Selection of external reactive power setpoint for frequency droop mode (above) *)
		rQ_Offs_Input := rQset_Droop;
	END_IF;

	rQ_Droop_Offs := LIMIT(Para.rQ_UnderExc_Lim * Para.rS_Nom, rQ_Offs_Input * Para.rS_Nom, Para.rQ_OverExc_Lim * Para.rS_Nom);	(* limit input *)

	VIS2MM.rQ_Droop_Set_Man	:= rQ_Droop_Offs / MAX(1.0,Para.rS_Nom);	(* set current setpoint to manual input, for smooth transition *)
	MM2VIS.rQ_Droop_Offs	:= rQ_Droop_Offs / MAX(1.0,Para.rS_Nom);

	(** U.1.4: calculate from Q offset to U offset *)
	rU_Droop_Offs := rQ_Droop_Offs / MAX(1.0,Para.rS_Nom) * Para.rU_StCtr_Grad;

	(** U.2: scale block for voltage droop *)
	xLCRScal_U_WPt.x  := IN_GC.tQ_Act[1].Ai;
	xLCRScal_U_WPt.x1 := -Para.rS_Nom;
	xLCRScal_U_WPt.x2 := Para.rS_Nom;
	xLCRScal_U_WPt.y1 := 1.0 + Para.rU_StCtr_Grad + rU_Droop_Offs;
	xLCRScal_U_WPt.y2 := 1.0 - Para.rU_StCtr_Grad + rU_Droop_Offs;
	xLCRScal_U_WPt();

	(** U.3: choose setpoint *)
	CASE iSrc_U_OffsSet OF
		0: xLCRRamp_U_Set_Norm.x := 1.0;					(* deactivated *)
		1: xLCRRamp_U_Set_Norm.x := xLCRScal_U_WPt.y;		(* Reactive power setpoint for droop curve *)
		2: xLCRRamp_U_Set_Norm.x := rUset_Isl;				(* Voltage setpoint *)
	END_CASE

	(** U.4: set point ramp 1%/s *)
	xLCRRamp_U_Set_Norm.enable	:= TRUE;
	xLCRRamp_U_Set_Norm.set		:= FALSE; 				(* always activate *)
	xLCRRamp_U_Set_Norm.y_set	:= 1.0;					(* if deactivated set to 100% *)
	xLCRRamp_U_Set_Norm.dy_up	:= 0.01;				(* ramp speed 1%/s *)
	xLCRRamp_U_Set_Norm.dy_down	:= 0.01;				(* ramp speed 1%/s *)
	xLCRRamp_U_Set_Norm.y_max	:= 1.10; 				(* max limit: 110%Unom *)
	xLCRRamp_U_Set_Norm.y_min	:= 0.90;				(* min limit:  90%Unom *)
	xLCRRamp_U_Set_Norm();
	IF NOT xOpMode.Island AND IN_GC.bU_Set_NP_Rel THEN	(* switch over setpoint without ramp for fast reaction *)
		OUT_GC.tU_Set_Norm.Ao := IN_GC.rU_Set_NP; 		(* mains parallel operation *)
	ELSE
		OUT_GC.tU_Set_Norm.Ao := xLCRRamp_U_Set_Norm.y;	(* island operation *)
	END_IF;

	(** U.5: Window size *)
	rQ_Win	:=	INT_TO_REAL(REAL_TO_INT(Para.rS_Nom) - (REAL_TO_INT(Para.rS_Nom) MOD 100) + 100);
	x_Win[0] :=	-rQ_Win;
	x_Win[1] :=	rQ_Win;
	MM2VIS.tU_Stat.tWin.x    := x_Win;
	MM2VIS.tU_Stat.tWin.y[0] := Para.rU_Gen_Nom[1] * 0.875;
	MM2VIS.tU_Stat.tWin.y[1] := Para.rU_Gen_Nom[1] * 1.125;

	(** U.6: Green line: Unom *)
	MM2VIS.tU_Stat.tLn_Nom.x	:= x_Win;
	MM2VIS.tU_Stat.tLn_Nom.y[0]	:= Para.rU_Gen_Nom[1];
	MM2VIS.tU_Stat.tLn_Nom.y[1]	:= Para.rU_Gen_Nom[1];

	(** U.7: Blue line: Uset *)
	MM2VIS.tU_Stat.tLn_Set.x[0]	:= -Para.rS_Nom;
	MM2VIS.tU_Stat.tLn_Set.x[1]	:= Para.rS_Nom;

	CASE iSrc_U_OffsSet OF
		0: 	MM2VIS.tU_Stat.tLn_Set.y[0]	:= Para.rU_Gen_Nom[1];
			MM2VIS.tU_Stat.tLn_Set.y[1]	:= Para.rU_Gen_Nom[1];

		1:	MM2VIS.tU_Stat.tLn_Set.y[0]	:= Para.rU_Gen_Nom[1] * (1.0 - MM2VIS.tU_Stat.tLn_Set.x[0] / MAX(1.0,Para.rS_Nom) * Para.rU_StCtr_Grad + rU_Droop_Offs);
			MM2VIS.tU_Stat.tLn_Set.y[1]	:= Para.rU_Gen_Nom[1] * (1.0 - MM2VIS.tU_Stat.tLn_Set.x[1] / MAX(1.0,Para.rS_Nom) * Para.rU_StCtr_Grad + rU_Droop_Offs);

		2:	MM2VIS.tU_Stat.tLn_Set.y[0]	:= Para.rU_Gen_Nom[1] * LIMIT(xLCRRamp_U_Set_Norm.y, 0.9, 1.1);
			MM2VIS.tU_Stat.tLn_Set.y[1]	:= Para.rU_Gen_Nom[1] * LIMIT(xLCRRamp_U_Set_Norm.y, 0.9, 1.1);
	END_CASE

	(** U.8: Brown point: Working point *)
	MM2VIS.tU_Stat.tWPt.x := LIMIT(IN_GC.tQ_Act[1].Ai, -rQ_Win, rQ_Win);
	MM2VIS.tU_Stat.tWPt.y := IN_GC.tU_Avg[1].Ai;

END_PROGRAM
```

#### v_ctr.var
```iecst
VAR
	bU_SyD_Inc : BOOL;
	bU_SyD_Dec : BOOL;
	rU_Gen_Diff_Match_p : REAL := 0.0; (*U offset leistungsabhängig*)
	rU_Gen_Diff_Match_sy : REAL := 0.0; (*U offset während SY*)
	rU_SY_diff : REAL; (*Voltage difference at SY*)
	rU_SY_span : REAL; (*Dead band voltage controller*)
	u_minus : BOOL; (*Voltage matching decreasing*)
	u_offset : REAL; (*U offset gesamt*)
	u_offset_f : REAL; (*U offset frequenzabhängig*)
	u_plus : BOOL; (*Voltage matching increasing*)
	U_TAKT : BOOL; (*Takt for voltage adjustment*)
	xRAMPE_rU_Gen_Diff_Match_p : RAMPE_R;
	xRAMPE_rU_Gen_Diff_Match_sy : RAMPE_R;
	xRAMPE_u_offset_f : RAMPE_R;
	xSigScal_u_offset_mA : xSigScal_R;
	xSigScal_u_offset_V : xSigScal_R;
	xSigScal_uoffset_f : xSigScal_R;
	xSigScal_uoffset_p : xSigScal_R;
	xTOF_Synch : TOF;
	xTON_U_TAKT : TON;
	xTON_U_TAKT_P : TON;
	xTP_U_DOWN : TP;
	xTP_U_UP : TP;
	xR_TRIG_u_plus : R_TRIG;
	xR_TRIG_u_minus : R_TRIG;
	rF_Act_norm : REAL;
	rU_diff_percent : REAL;
	tiPuls : TIME;
	x_Win : ARRAY[0..1] OF REAL; (* window on HMI: max & min values for x&y *)
	rQ_Nom : REAL; (* max reactive power [kVAr] *)
	xLCRScal_U_WPt : LCRScal; (* reactive power x [kVAr], voltage setpoint y [%Unom] *)
	xLCRRamp_U_Set_Norm : LCRRamp; (* Ramp to fade in [%Unom] *)
	iSrc_U_OffsSet : INT := 0; (*Voltage offset set point in island mode: 0= no setpoint, 1= Droop, 2= External *)
	rP_Nom_PF08 : REAL := 0.0;
	rQ_Offs_Input : REAL := 0.0;
	rU_Droop_Offs : REAL := 0.0;
	rQ_Droop_Offs : REAL := 0.0;
	rBuffer_U_SetExt : ARRAY[0..10] OF REAL;
	z_U_SetExt : INT;
	x_U_SetExt : INT;
	xTON_GoodQual_U_SetExt : TON;
	rLCRLimScal_U_SetExt_old : REAL;
	bBuffer_U_SetExt : BOOL := 0;
	rU_setExt : REAL; (* Skalierter Wert AI:U Sollwert von extern [V] *)
	rUset_Isl : REAL;
	bUset_Isl : BOOL;
	rBuffer_Q_Droop_Set : ARRAY[0..10] OF REAL;
	z_Q_Droop_Set : INT;
	x_Q_Droop_Set : INT;
	xTON_GoodQual_Q_Droop_Set : TON;
	rLCRLimScal_Q_Droop_Set_old : REAL;
	bBuffer_Q_Droop_Set : BOOL := 0;
	rQ_Droop_SetExt : REAL; (* Skalierter Wert AI:U Sollwert von extern [V] *)
	rQset_Droop : REAL;
	bQset_Droop : BOOL;
	rQ_Win : REAL;
END_VAR
```

### Program Logical/Generator/Ctr_GenPF (IEC, version 4.11.0) - power factor controller, not used

#### Ctr_GenPFCyclic.st
```iecst
(********************************************************************
Ctr_GenPF	 			 Generator cosphi controller

This code is confidential AND proprietary to the INNIO Company.
It may NOT be used in any form, or reproduced in any manner,
without written permission of the INNIO Company.
Copyright, INNIO Company, 2022

Customized modifications: -
------------------------

History:
-------
4.00.00	01.01.2013	ganguly		new
4.00.01	16.05.2014	lettenb.	controller release-bugfix, cleanup
4.00.02	21.05.2014	lettenb.	controller y.set, bugfix
		04.06.2014				controller .Y_set_Active IF gridcode is active, bugfix
4.00.03 28.01.2015 	lettenb.	task renamed: Ctr_Gen_13 -> Ctr_GenPF
V4.09.0	03.02.2020	lettenb.	autotune enabled, bugfix
V4.11.0	28.01.2022	Perktold	included plant controller upgrade

Instructions for use: -
--------------------

Outstandings:
------------

*******************************************************************************)

PROGRAM _CYCLIC

IF Para.bCtrGenPF_Active THEN

	(* Parameter Generator controller 13 *)
	Para.tCtrGenPF.W_set;
	Para.tCtrGenPF.W_set2;
	Para.tCtrGenPF.W_min;
	Para.tCtrGenPF.W_max;
	Para.tCtrGenPF.dW_up;
	Para.tCtrGenPF.dW_down;
	Para.tCtrGenPF.deadband;
	Para.tCtrGenPF.Y_min;
	Para.tCtrGenPF.Y_max;
	Para.tCtrGenPF.dY_max;
	Para.tCtrGenPF.Y_block;
	Para.tCtrGenPF.invert;
	Para.tCtrGenPF.Kp;
	Para.tCtrGenPF.Tn;
	Para.tCtrGenPF.Tv;
	Para.tCtrGenPF.Kp_GainScheduling;
	Para.tCtrGenPF.Tn_GainScheduling;
	Para.tCtrGenPF.Tv_GainScheduling;
	Para.tCtrGenPF.t_min_pulse_down;
	Para.tCtrGenPF.t_min_pulse_up;
	Para.tCtrGenPF.t_period_down;
	Para.tCtrGenPF.t_period_up;

	(* Input variable *)
	tCtrGenPF_In := VIS2MM.tCtrGenPF_In;	(* from vis *)

	(* Input from module *)
	tCtrGenPF_In.enable		  	:= 	Para.bPF_CosPCtr_Ena
							AND NOT OUT_GC.bPF_CosPCtr_block
							AND 	IN_GC.tPB2MM.bParaSetupOk;
	tCtrGenPF_In.W_ext_Active	:=	tCtrGenPF_In.W_ext_Active OR TRUE;	(* no changeover to internal *)
	tCtrGenPF_In.W_ext		 	:=	PFSoll_lin;  						(* linearised PF_Soll_value  *)
	tCtrGenPF_In.Y_set_Active	:= (IN_GC.bGCQ_Fun_Act OR Para.bPF_CosPCtr_Ena)
								AND OUT_GC.bPF_CosPCtr_block;			(* depending on operating mode *)
	tCtrGenPF_In.Y_set		 	:=	OUT_GC.rPF_CosPCtr_block;			(* depending on operating mode *)
	IF xOpMode.NetP THEN
		tCtrGenPF_In.X			:=	PF_Ist_lin; 						(* linearised PF_Ist_value, power factor process value (actual)*)
	ELSE
		tCtrGenPF_In.X			:=	1.0; 								(* freeze linearised PF_Ist_value for visu, power factor process value (actual)*)
	END_IF;
	tCtrGenPF_In.A			 	:=	0.0;
	tCtrGenPF_In.W_set2_Active	:= FALSE;		(*Input to define which internal setpoint will be used TRUE = use the 2nd set point | FALSE use the normal "1st" one*)
	tCtrGenPF_In.GainScheduling	:= 0.0;			(*Input for Gain Scheduling: 0.0 = use 100% of the Standard PID-Parameters | 1.0 = use 100% of the GainSched. PID Parameters | linear interpolation in between*)
	tCtrGenPF_In.Y_min_cust		:= -1.0;		(*"customized" Y-Min at the current moment (The existing Y-Min parameter is the global minimum. To have an effect Y_min_cust needs to be > the parameter | -1.0 = function not used*)
	tCtrGenPF_In.Y_max_cust		:= 1.0;			(*"customized" Y-Max at the current moment (The existing Y-Max parameter is the global maximum. To have an effect Y_max_cust needs to be < the parameter | 1.0 = function not used*)
	tCtrGenPF_In.Retrigger		:= FALSE;		(*a rising edge on this input signals the controller to retrigger - set W on X and force the Integrator to the current Y*)

	(* Input from Visualization via OPC *)
	tCtrGenPF_In.Y_man_Active;
	tCtrGenPF_In.Y_man;
	tCtrGenPF_In.X_min;
	tCtrGenPF_In.X_max;
	tCtrGenPF_In.Tune_quality;
	tCtrGenPF_In.Tune_PI;
	tCtrGenPF_In.Tune_PID;
	tCtrGenPF_In.Tune_start;
	tCtrGenPF_In.Tune_stop;
	tCtrGenPF_In.Tune_takeover;

	xCtrGenPF();

	(* Output variables  Generator controller 13 function block *)
	(* Output to module(s) *)
	OUT_GC.rCtrGenPF_Set := tCtrGenPF_Out.Y;			//Analog OUT (-100..100%)

	(* Output to Visualization via OPC *)
	MM2VIS.tCtrGenPF_Out := tCtrGenPF_Out;
	VIS2MM.tCtrGenPF_In  := tCtrGenPF_In;

	tCtrGenPF_Out.Active;
	tCtrGenPF_Out.Y;
	tCtrGenPF_Out.W;
	tCtrGenPF_Out.e;
	tCtrGenPF_Out.Kp_tune;
	tCtrGenPF_Out.Tn_tune;
	tCtrGenPF_Out.Tv_tune;
	tCtrGenPF_Out.status;

ELSE
	(* Set OUT values to 0 in case of Controller is not active *)

	OUT_GC.rCtrGenPF_Set   	       := Para.tCtrGenPF.Y_block;

	tCtrGenPF_Out.Active;
	tCtrGenPF_Out.Y;
	tCtrGenPF_Out.W;
	tCtrGenPF_Out.e;
	tCtrGenPF_Out.Kp_tune;
	tCtrGenPF_Out.Tn_tune;
	tCtrGenPF_Out.Tv_tune;
	tCtrGenPF_Out.status;

END_IF;

END_PROGRAM
```

#### Ctr_GenPFInit.st
```iecst
(********************************************************************
 * COPYRIGHT -- INNIO Company
 ********************************************************************
 * Program: CtrGenPF
 * File: CtrGenPFInit.st
 * Author: 105051626
 * Created: January 08, 2013
 ********************************************************************
 * Implementation of program CtrGenPF
 ********************************************************************)

PROGRAM _INIT

	(*Parameter FACTORY DEFAULT VALUES *)
	(*for missing/new/not visualized parameter*)
	Para.tCtrGenPF.t_min_pulse_down  := 10;
	Para.tCtrGenPF.t_min_pulse_up	 := 10;
	Para.tCtrGenPF.t_period_down	 := 100;
	Para.tCtrGenPF.t_period_up	     := 100;
	VIS2MM.tCtrGenPF_In.W_ext_Active := TRUE;  // Generator controller is programmed to use the W_Set (external set point) input
											   // It does not use the X_Set (internal set points) inputs

	Para.tCtrGenPF.Y_block          := 0.25;   // Force output to 0,25 from controller when disabled.

	tCtrGenPF_In.AlwaysUseYRamp		:= TRUE;	(*If TRUE the Y signal will always limit the change rate via the according parameter | if FALSE the Y signal will jump in case the controller is disabled (blocked or set)*)
	tCtrGenPF_In.KeepYManAtBlock	:= TRUE;	(*If TRUE the controller will keep the Y-man value constant in case the controller is disabled (blocked or set) | If FALSE the blocked or set value will override the Y-man value*)
	tCtrGenPF_In.Y_min_cust			:= -1.0;	(*"customized" Y-Min at the current moment (The existing Y-Min parameter is the global minimum. To have an effect Y_min_cust needs to be > the parameter | -1.0 = function not used*)
	tCtrGenPF_In.Y_max_cust			:=  1.0;	(*"customized" Y-Max at the current moment (The existing Y-Max parameter is the global maximum. To have an effect Y_max_cust needs to be < the parameter | 1.0 = function not used*)
	tCtrGenPF_In.StepperMode		:= FALSE;	(* TRUE = use PWM-Mode (standard mode until 4.10) | FALSE = use continuous servo drive *)

	xCtrGenPF.pParameter := ADR(Para.tCtrGenPF);
	xCtrGenPF.pInput     := ADR(tCtrGenPF_In);
	xCtrGenPF.pOutput    := ADR(tCtrGenPF_Out);

END_PROGRAM
```

### Program Logical/Generator/Ctr_Q (IEC, version 4.11.0) - reactive power controller

#### Ctr_QCyclic.st
```iecst
(********************************************************************
Ctr_Q		reactive power controller

This code is confidential AND proprietary to the INNIO Company.
It may NOT be used in any form, or reproduced in any manner,
without written permission of the INNIO Company.
Copyright, INNIO Company, 2022

Customized modifications: -
------------------------

History:
-------
V4.05.0	21.11.2017 	lettenb.	new, GR redesign, PF control -> Q control
V4.09.0	19.11.2019	lettenb.	ctr freeze conditions added
		03.02.2020	lettenb.	autotune enabled, bugfix
V4.10.0 18.01.2021	Weitzer		OUT_GC.tCtr_Q_Out interface for Customized added - AB specific
V4.11.0	28.01.2022	Perktold	included plant controller upgrade

Instructions for use: -
--------------------

Outstandings:
------------

*******************************************************************************)

PROGRAM _CYCLIC

	(* Parameter reactive power controller 33 *)
	Para.tCtr_Q.W_set;
	Para.tCtr_Q.W_set2;
	Para.tCtr_Q.W_min;
	Para.tCtr_Q.W_max;
	Para.tCtr_Q.dW_up;
	Para.tCtr_Q.dW_down;
	Para.tCtr_Q.deadband;
	Para.tCtr_Q.Y_min;
	Para.tCtr_Q.Y_max;
	Para.tCtr_Q.dY_max;
	Para.tCtr_Q.Y_block;
	Para.tCtr_Q.invert;
	Para.tCtr_Q.Kp;
	Para.tCtr_Q.Tn;
	Para.tCtr_Q.Tv;
	Para.tCtr_Q.Kp_GainScheduling;
	Para.tCtr_Q.Tn_GainScheduling;
	Para.tCtr_Q.Tv_GainScheduling;
	Para.tCtr_Q.t_min_pulse_down;
	Para.tCtr_Q.t_min_pulse_up;
	Para.tCtr_Q.t_period_down;
	Para.tCtr_Q.t_period_up;

	(* Input variable *)
	tCtr_Q_In := VIS2MM.tCtr_Q_In;	(* from vis *)

	(* Input from module *)
	tCtr_Q_In.enable	 	:=  Para.bPF_CosPCtr_Ena
						AND		Para.bCtr_Q
						AND NOT(Para.iQ_GrC_PointCtrl = 3)				(* direct control *)
						AND NOT OUT_GC.bPF_CosPCtr_block
						AND 	IN_GC.tPB2MM.bParaSetupOk;
	tCtr_Q_In.W_ext_Active	:=	tCtr_Q_In.W_ext_Active OR TRUE;			(* no changeover to internal *)
	tCtr_Q_In.W_ext		 	:=	rQ_Set_Lim;

	IF Para.bPF_CosPCtr_Ena AND OUT_GC.bPF_CosPCtr_block THEN			(* depending on operating mode *)
		tCtr_Q_In.Y_set_Active	:=  TRUE;
		tCtr_Q_In.Y_set		 	:=	OUT_GC.rPF_CosPCtr_block;
	ELSIF IN_GC.bMsg2831 												(* freeze ctr depending on FRT event *)
	  OR (IN_GC.tU_Avg[1].Ai < (Para.rU_Gen_Nom[1] * 0.85))				(* measured voltage of MMU is below 85% *)
	  OR (MM2VIS.rQ_AVR_Set_Norm >= Para.rQ_UnderExc_Lim)				(* Q_AVR_Set = limit *)// AVR_Lim grenzen erhöhen um reglerhub an den grenzen zu ermöglichen - lukas?
	  OR (MM2VIS.rQ_AVR_Set_Norm <= Para.rQ_OverExc_Lim) THEN                                  // AVR_Lim grenzen erhöhen um reglerhub an den grenzen zu ermöglichen - lukas?
		tCtr_Q_In.Y_set_Active	:=  TRUE;
		tCtr_Q_In.Y_set		 	:=	tCtr_Q_Out.Y;						(* freeze actual y *)
	ELSE
		tCtr_Q_In.Y_set_Active	:=  FALSE;
	END_IF;

	(* calculation Qact from voltage POC *)
	(* Qact[%] = ( Uact[V] * 100 / Unom_par.11696[V] ) - 100; *)
	IF Para.rU_GrC_SetEU_Nom > 0 THEN
		rQ_POC_Act_CalcV := 2.0 * ((rU_POC_Act / Para.rU_GrC_SetEU_Nom) - 1); (* 2.0 = factor to get higher controller deviation *)
	END_IF;

	IF xOpMode.NetP THEN
		IF Para.iQ_GrC_CtrlFun = 7 THEN	tCtr_Q_In.X := rQ_POC_Act_CalcV;(* V control *)
		ELSE			                tCtr_Q_In.X := rQ_POC_Act_Norm;	(* Q control *)
		END_IF;
	ELSE
		tCtr_Q_In.X := 0.0;
	END_IF;

	tCtr_Q_In.X; 							(* Q process value (actual) *)
	tCtr_Q_In.A			 	:=	0.0;
	tCtr_Q_In.W_set2_Active	:= FALSE;		(*Input to define which internal setpoint will be used TRUE = use the 2nd set point | FALSE use the normal "1st" one*)
	tCtr_Q_In.GainScheduling:= 0.0;			(*Input for Gain Scheduling: 0.0 = use 100% of the Standard PID-Parameters | 1.0 = use 100% of the GainSched. PID Parameters | linear interpolation in between*)
	tCtr_Q_In.Y_min_cust	:= -1.0;		(*"customized" Y-Min at the current moment (The existing Y-Min parameter is the global minimum. To have an effect Y_min_cust needs to be > the parameter | -1.0 = function not used*)
	tCtr_Q_In.Y_max_cust	:= 1.0;			(*"customized" Y-Max at the current moment (The existing Y-Max parameter is the global maximum. To have an effect Y_max_cust needs to be < the parameter | 1.0 = function not used*)
	tCtr_Q_In.Retrigger		:= FALSE;		(*a rising edge on this input signals the controller to retrigger - set W on X and force the Integrator to the current Y*)

	(* Input from Visualization via OPC *)
	tCtr_Q_In.Y_man_Active;
	tCtr_Q_In.Y_man;
	tCtr_Q_In.X_min;
	tCtr_Q_In.X_max;
	tCtr_Q_In.Tune_quality;
	tCtr_Q_In.Tune_PI;
	tCtr_Q_In.Tune_PID;
	tCtr_Q_In.Tune_start;
	tCtr_Q_In.Tune_stop;
	tCtr_Q_In.Tune_takeover;

	xCtr_Q();

	(* Output variables function block *)
	(* Output to module(s) *)
	OUT_GC.rCtr_Q_Set := tCtr_Q_Out.Y;	(* controller out -1,0..0..+1,0 = -100%Qnom..0..+100%Qnom *)
	OUT_GC.tCtr_Q_Out := tCtr_Q_Out;	(* Interface for Customized - AB Specific *)

	(* Output to Visualization via OPC *)
	MM2VIS.tCtr_Q_Out := tCtr_Q_Out;
	VIS2MM.tCtr_Q_In  := tCtr_Q_In;		(* write back to IN_struct for reset: Tune_takeover, X-display, ...!*)

	tCtr_Q_Out.Active;
	tCtr_Q_Out.Y;
	tCtr_Q_Out.W;
	tCtr_Q_Out.e;
	tCtr_Q_Out.Kp_tune;
	tCtr_Q_Out.Tn_tune;
	tCtr_Q_Out.Tv_tune;
	tCtr_Q_Out.status;

END_PROGRAM
```

#### Ctr_QInit.st
```iecst
PROGRAM _INIT

	xCtr_Q.pParameter := ADR(Para.tCtr_Q);
	xCtr_Q.pInput     := ADR(tCtr_Q_In);
	xCtr_Q.pOutput    := ADR(tCtr_Q_Out);

	tCtr_Q_In.AlwaysUseYRamp		:= TRUE;	(*If TRUE the Y signal will always limit the change rate via the according parameter | if FALSE the Y signal will jump in case the controller is disabled (blocked or set)*)
	tCtr_Q_In.KeepYManAtBlock		:= TRUE;	(*If TRUE the controller will keep the Y-man value constant in case the controller is disabled (blocked or set) | If FALSE the blocked or set value will override the Y-man value*)
	tCtr_Q_In.Y_min_cust			:= -1.0;	(*"customized" Y-Min at the current moment (The existing Y-Min parameter is the global minimum. To have an effect Y_min_cust needs to be > the parameter | -1.0 = function not used*)
	tCtr_Q_In.Y_max_cust			:=  1.0;	(*"customized" Y-Max at the current moment (The existing Y-Max parameter is the global maximum. To have an effect Y_max_cust needs to be < the parameter | 1.0 = function not used*)
	tCtr_Q_In.StepperMode			:= FALSE;	(* TRUE = use PWM-Mode (standard mode until 4.10) | FALSE = use continuous servo drive *)

END_PROGRAM
```

### Program Logical/Generator/gen_aux (IEC, version 4.11.0) - generator auxiliaries

#### gen_auxCyclic.st
```iecst
(*******************************************************************************
gen_aux		generator auxiliaries

This code is confidential and proprietary to the INNIO Company.
It may not be used in any form, or reproduced in any manner,
without the express written permission of the INNIO Company.
Copyright, INNIO Company, 2022

Customized modifications: -
------------------------

History:
-------
V3.40.0	22.11.2011	lettenb.	new
V3.99.9 13.02.2014  ganguly     modified Generator preheating condition changed because
								Generator PTC monitoring -> Standstill heating OF generator
								does not shut off.
V4.01.0 19.05.2014	Denk		Generator preheating condition changed IN_GC.tECW_PreH_Dem.Do;
V4.01.1	12.02.2014	lettenb.	Genoheizung von Vorwärmpumpe trennen, Vorwärmpumpe wird auch für hydraulische
								Vorwärmung und/oder für Abkühlprogramm verwendet (920 stapelfeld)
V4.04.0	18.05.2016	lettenb.	DO_GEN_BERC added from ex task gen_lub: demand lubeoil cooling system, bugfix
V4.05.0 30.03.2017	lettenb.	xGR_MAX_GenPreH.Gw: - 0.5, Hy:= 0.5 =>  - 5.0, Hy:= 5.0, bugfix
V4.07.0	29.04.2019	lettenb.	1054 fire alarm added(separation from safety loop(1031) with safety PLC)
		30.07.2019	lettenb.	LOS_Dem.Do: 1054,1031 added(safety request, doujak andreas) bu01
V4.11.0	05.11.2021	Schmid		Generator preheating independent of electric or hydraulic ECW preheating
		18.01.2022	lettenb.	generator bearing lubrication(Aerotherm) demand for bN2_ScavCoPrelubeOn OR IN_GC.bEO_PrelubeDemIgn, bugfix

Instructions for use:
--------------------
Outstandings:
------------
*******************************************************************************)

PROGRAM _CYCLIC

	(*------------------------------------------------------------------------------------*)
	(* generator preheating *)
	xGR_MAX_GenPreH(In:= IN_GC.tT_Gen_Bear_B_Act.Ai, Gw:= Para.rT_Gen_Bear_Lim_B - 5.0, Hy:= 5.0);	(* NDE bearing temperature *)
	xTON_MAX_GenPreH(IN:= xGR_MAX_GenPreH.Q, PT:= T#2s);

	IF xEngType.Type9 THEN 				OUT_GC.tGen_PreHDem.Do := bOMSS_MAT AND NOT IN_GC.bEng_Aux_Dem_CDR AND NOT IN_GC.bMsg1031 AND NOT IN_GC.bMsg1054 AND NOT xTON_MAX_GenPreH.Q;
	ELSIF Para.bT_Gen_Bear_B_Ena THEN	OUT_GC.tGen_PreHDem.Do := IN_GC.tECWP_PreH_Dem.Do AND NOT xTON_MAX_GenPreH.Q;
	ELSE								OUT_GC.tGen_PreHDem.Do := IN_GC.bECW_Gnl_PreH_Dem;
	END_IF;

	(*------------------------------------------------------------------------------------*)
	(* generator: demand (aerotherm) lubeoil/cooling system LSA56, TD125, WD130 (not 920) *)
    OUT_GC.tLOS_Dem.Do := (IN_GC.bEng_Aux_Dem OR M_DREHZ OR IN_GC.bN2_ScavCoPrelubeOn OR IN_GC.bEO_PrelubeDemIgn)
				   AND NOT IN_GC.bMsg1031
				   AND NOT IN_GC.bMsg1054;

END_PROGRAM
```

#### gen_aux.var
```iecst
(********************************************************************
 * COPYRIGHT -- INNIO Company
 ********************************************************************
 * Program: gen_aux
 * File: gen_aux.var
 * Author: 105051626
 * Created: March 19, 2013
 ********************************************************************
 * Local variables of program gen_aux
 ********************************************************************)
VAR
	xGR_MAX_GenPreH : GR_MAXR;
	xTON_MAX_GenPreH : TON;
END_VAR
```

### Program Logical/Generator/oilskid (IEC, version 4.10.0) - oilskid
